SPLINE
SPL {X  -151.875, Y  +721.838, Z    +0.000, E1   -27.241, E3 +55166.889}
SPL {X  -157.803, Y  +697.921, Z    +0.000, E1   -15.861, E3 +55182.756}
SPL {X  -159.710, Y  +681.128, Z    +0.000, E1    -6.465, E3 +55187.890}
SPL {X  -159.999, Y  +671.996, Z    +0.000, E1    -0.411, E3 +55189.220}
SPL {X  -160.000, Y  +665.132, Z    +0.000, E1    +5.902, E3 +55190.030}
SPL {X  -160.000, Y  +655.952, Z    +0.000, E1   +16.601, E3 +55192.025}
SPL {X  -160.000, Y  +643.612, Z    +0.000, E1   +29.091, E3 +55196.997}
SPL {X  -160.000, Y  +606.346, Z    +0.000, E1   +46.235, E3 +55224.805}
SPL {X  -160.000, Y  +564.751, Z    +0.000, E1   +49.682, E3 +55279.976}
SPL {X  -160.000, Y  +555.844, Z    +0.000, E1   +49.673, E3 +55296.057}
SPL {X  -160.000, Y  +545.889, Z    +0.000, E1   +49.702, E3 +55313.956}
SPL {X  -160.000, Y  +535.482, Z    +0.000, E1   +49.684, E3 +55332.755}
SPL {X  -160.000, Y  +526.440, Z    +0.000, E1   +49.666, E3 +55349.088}
SPL {X  -160.000, Y  +518.889, Z    +0.000, E1   +49.624, E3 +55362.913}
ENDSPLINE

SPLINE
SPL {X  -160.000, Y  +548.948, Z    +0.000, E1   +36.551, E3 +55372.601}
ENDSPLINE

SPLINE
SPL {X  -160.000, Y  +541.880, Z    +0.000, E1   +37.562, E3 +55386.380}
SPL {X  -160.000, Y  +532.200, Z    +0.000, E1   +38.842, E3 +55404.721}
SPL {X  -160.000, Y  +523.085, Z    +0.000, E1   +39.970, E3 +55421.412}
SPL {X  -160.000, Y  +513.603, Z    +0.000, E1   +41.139, E3 +55437.996}
SPL {X  -160.000, Y  +503.235, Z    +0.000, E1   +42.462, E3 +55454.704}
SPL {X  -160.000, Y  +493.516, Z    +0.000, E1   +43.493, E3 +55470.749}
SPL {X  -160.000, Y  +483.478, Z    +0.000, E1   +44.599, E3 +55486.207}
SPL {X  -160.000, Y  +473.020, Z    +0.000, E1   +45.665, E3 +55502.037}
SPL {X  -160.000, Y  +461.024, Z    +0.000, E1   +46.836, E3 +55519.512}
SPL {X  -160.000, Y  +448.988, Z    +0.000, E1   +48.043, E3 +55535.774}
SPL {X  -160.000, Y  +439.029, Z    +0.000, E1   +48.623, E3 +55551.181}
SPL {X  -160.000, Y  +429.710, Z    +0.000, E1   +48.622, E3 +55568.628}
SPL {X  -160.000, Y  +420.891, Z    +0.000, E1   +48.613, E3 +55585.153}
SPL {X  -160.000, Y  +412.565, Z    +0.000, E1   +48.611, E3 +55600.718}
SPL {X  -160.000, Y  +404.943, Z    +0.000, E1   +48.601, E3 +55615.021}
SPL {X  -160.000, Y  +395.837, Z    +0.000, E1   +48.634, E3 +55632.010}
SPL {X  -159.987, Y  +386.768, Z    +0.000, E1   +48.609, E3 +55649.015}
SPL {X  -159.620, Y  +377.782, Z    +0.000, E1   +48.569, E3 +55666.183}
SPL {X  -158.761, Y  +368.924, Z    +0.000, E1   +48.401, E3 +55683.710}
SPL {X  -157.560, Y  +360.964, Z    +0.000, E1   +48.177, E3 +55699.881}
SPL {X  -156.187, Y  +354.076, Z    +0.000, E1   +47.920, E3 +55714.214}
SPL {X  -154.507, Y  +347.236, Z    +0.000, E1   +47.623, E3 +55728.742}
SPL {X  -152.108, Y  +339.169, Z    +0.000, E1   +47.215, E3 +55746.219}
SPL {X  -149.264, Y  +331.177, Z    +0.000, E1   +46.657, E3 +55764.018}
SPL {X  -146.675, Y  +324.875, Z    +0.000, E1   +46.130, E3 +55778.371}
SPL {X  -140.793, Y  +312.792, Z    +0.000, E1   +40.077, E3 +55852.614}
ENDSPLINE

SPLINE
SPL {X  -154.674, Y  +347.860, Z    +0.000, E1   +23.016, E3 +55922.757}
SPL {X  -159.179, Y  +372.617, Z    +0.000, E1   +10.186, E3 +55935.406}
SPL {X  -159.924, Y  +383.861, Z    +0.000, E1    +3.320, E3 +55938.028}
SPL {X  -160.000, Y  +389.631, Z    +0.000, E1    -0.873, E3 +55938.744}
SPL {X  -160.000, Y  +394.628, Z    +0.000, E1    -5.657, E3 +55939.420}
SPL {X  -160.000, Y  +401.354, Z    +0.000, E1   -13.067, E3 +55940.811}
SPL {X  -160.000, Y  +413.710, Z    +0.000, E1   -25.976, E3 +55945.603}
SPL {X  -160.000, Y  +449.556, Z    +0.000, E1   -44.518, E3 +55971.645}
SPL {X  -160.000, Y  +494.814, Z    +0.000, E1   -49.280, E3 +56029.994}
SPL {X  -160.000, Y  +504.699, Z    +0.000, E1   -49.282, E3 +56048.074}
SPL {X  -160.000, Y  +515.266, Z    +0.000, E1   -49.291, E3 +56067.388}
SPL {X  -160.000, Y  +526.314, Z    +0.000, E1   -49.296, E3 +56087.617}
SPL {X  -160.000, Y  +536.842, Z    +0.000, E1   -49.263, E3 +56106.943}
SPL {X  -160.000, Y  +547.071, Z    +0.000, E1   -49.286, E3 +56125.620}
SPL {X  -160.000, Y  +558.279, Z    +0.000, E1   -49.288, E3 +56146.124}
SPL {X  -160.000, Y  +568.309, Z    +0.000, E1   -49.259, E3 +56164.519}
SPL {X  -160.000, Y  +579.695, Z    +0.000, E1   -49.320, E3 +56185.249}
SPL {X  -160.000, Y  +592.166, Z    +0.000, E1   -49.294, E3 +56208.109}
SPL {X  -160.000, Y  +603.260, Z    +0.000, E1   -49.285, E3 +56228.434}
SPL {X  -160.000, Y  +615.079, Z    +0.000, E1   -49.301, E3 +56250.046}
SPL {X  -160.000, Y  +627.012, Z    +0.000, E1   -49.289, E3 +56271.898}
SPL {X  -160.000, Y  +638.544, Z    +0.000, E1   -49.285, E3 +56293.009}
SPL {X  -160.000, Y  +649.673, Z    +0.000, E1   -49.278, E3 +56313.382}
SPL {X  -160.000, Y  +661.315, Z    +0.000, E1   -49.297, E3 +56334.652}
SPL {X  -159.993, Y  +672.984, Z    +0.000, E1   -49.282, E3 +56356.043}
SPL {X  -159.528, Y  +683.783, Z    +0.000, E1   -49.201, E3 +56376.297}
SPL {X  -158.288, Y  +694.841, Z    +0.000, E1   -49.005, E3 +56397.811}
SPL {X  -156.479, Y  +704.881, Z    +0.000, E1   -48.644, E3 +56418.125}
SPL {X  -154.000, Y  +714.904, Z    +0.000, E1   -48.243, E3 +56438.934}
SPL {X  -150.967, Y  +724.498, Z    +0.000, E1   -47.642, E3 +56459.599}
SPL {X  -147.384, Y  +733.774, Z    +0.000, E1   -47.000, E3 +56480.072}
SPL {X  -139.301, Y  +750.209, Z    +0.000, E1   -41.935, E3 +56551.253}
ENDSPLINE

SPLINE
SPL {X  -151.875, Y  +721.838, Z    +0.000, E1   -27.241, E3 +56628.423}
SPL {X  -157.803, Y  +697.921, Z    +0.000, E1   -15.861, E3 +56644.290}
SPL {X  -159.710, Y  +681.128, Z    +0.000, E1    -6.465, E3 +56649.424}
SPL {X  -159.999, Y  +671.996, Z    +0.000, E1    -0.411, E3 +56650.754}
SPL {X  -160.000, Y  +665.132, Z    +0.000, E1    +5.902, E3 +56651.564}
SPL {X  -160.000, Y  +655.952, Z    +0.000, E1   +16.601, E3 +56653.560}
SPL {X  -160.000, Y  +643.612, Z    +0.000, E1   +29.091, E3 +56658.531}
SPL {X  -160.000, Y  +606.346, Z    +0.000, E1   +46.235, E3 +56686.339}
SPL {X  -160.000, Y  +564.751, Z    +0.000, E1   +49.682, E3 +56741.511}
SPL {X  -160.000, Y  +555.844, Z    +0.000, E1   +49.673, E3 +56757.591}
SPL {X  -160.000, Y  +545.889, Z    +0.000, E1   +49.702, E3 +56775.490}
SPL {X  -160.000, Y  +535.482, Z    +0.000, E1   +49.684, E3 +56794.289}
SPL {X  -160.000, Y  +526.440, Z    +0.000, E1   +49.666, E3 +56810.623}
SPL {X  -160.000, Y  +518.889, Z    +0.000, E1   +49.624, E3 +56824.447}
ENDSPLINE

SPLINE
SPL {X  -160.000, Y  +548.948, Z    +0.000, E1   +36.551, E3 +56834.136}
ENDSPLINE

SPLINE
SPL {X  -160.000, Y  +541.880, Z    +0.000, E1   +37.562, E3 +56847.914}
SPL {X  -160.000, Y  +532.200, Z    +0.000, E1   +38.842, E3 +56866.255}
SPL {X  -160.000, Y  +523.085, Z    +0.000, E1   +39.970, E3 +56882.946}
SPL {X  -160.000, Y  +513.603, Z    +0.000, E1   +41.139, E3 +56899.530}
SPL {X  -160.000, Y  +503.235, Z    +0.000, E1   +42.462, E3 +56916.238}
SPL {X  -160.000, Y  +493.516, Z    +0.000, E1   +43.493, E3 +56932.283}
SPL {X  -160.000, Y  +483.478, Z    +0.000, E1   +44.599, E3 +56947.741}
SPL {X  -160.000, Y  +473.020, Z    +0.000, E1   +45.665, E3 +56963.571}
SPL {X  -160.000, Y  +461.024, Z    +0.000, E1   +46.836, E3 +56981.046}
SPL {X  -160.000, Y  +448.988, Z    +0.000, E1   +48.043, E3 +56997.308}
SPL {X  -160.000, Y  +439.029, Z    +0.000, E1   +48.623, E3 +57012.715}
SPL {X  -160.000, Y  +429.710, Z    +0.000, E1   +48.622, E3 +57030.162}
SPL {X  -160.000, Y  +420.891, Z    +0.000, E1   +48.613, E3 +57046.687}
SPL {X  -160.000, Y  +412.565, Z    +0.000, E1   +48.611, E3 +57062.253}
SPL {X  -160.000, Y  +404.943, Z    +0.000, E1   +48.601, E3 +57076.555}
SPL {X  -160.000, Y  +395.837, Z    +0.000, E1   +48.634, E3 +57093.545}
SPL {X  -159.987, Y  +386.768, Z    +0.000, E1   +48.609, E3 +57110.549}
SPL {X  -159.620, Y  +377.782, Z    +0.000, E1   +48.569, E3 +57127.717}
SPL {X  -158.761, Y  +368.924, Z    +0.000, E1   +48.401, E3 +57145.244}
SPL {X  -157.560, Y  +360.964, Z    +0.000, E1   +48.177, E3 +57161.415}
SPL {X  -156.187, Y  +354.076, Z    +0.000, E1   +47.920, E3 +57175.748}
SPL {X  -154.507, Y  +347.236, Z    +0.000, E1   +47.623, E3 +57190.276}
SPL {X  -152.108, Y  +339.169, Z    +0.000, E1   +47.215, E3 +57207.753}
SPL {X  -149.264, Y  +331.177, Z    +0.000, E1   +46.657, E3 +57225.552}
SPL {X  -146.675, Y  +324.875, Z    +0.000, E1   +46.130, E3 +57239.905}
SPL {X  -140.793, Y  +312.792, Z    +0.000, E1   +40.077, E3 +57314.148}
ENDSPLINE

SPLINE
SPL {X  -154.674, Y  +347.860, Z    +0.000, E1   +23.016, E3 +57384.291}
SPL {X  -159.179, Y  +372.617, Z    +0.000, E1   +10.186, E3 +57396.940}
SPL {X  -159.924, Y  +383.861, Z    +0.000, E1    +3.320, E3 +57399.562}
SPL {X  -160.000, Y  +389.631, Z    +0.000, E1    -0.873, E3 +57400.278}
SPL {X  -160.000, Y  +394.628, Z    +0.000, E1    -5.657, E3 +57400.954}
SPL {X  -160.000, Y  +401.354, Z    +0.000, E1   -13.067, E3 +57402.345}
SPL {X  -160.000, Y  +413.710, Z    +0.000, E1   -25.976, E3 +57407.137}
SPL {X  -160.000, Y  +449.556, Z    +0.000, E1   -44.518, E3 +57433.179}
SPL {X  -160.000, Y  +494.814, Z    +0.000, E1   -49.280, E3 +57491.529}
SPL {X  -160.000, Y  +504.699, Z    +0.000, E1   -49.282, E3 +57509.608}
SPL {X  -160.000, Y  +515.266, Z    +0.000, E1   -49.291, E3 +57528.922}
SPL {X  -160.000, Y  +526.314, Z    +0.000, E1   -49.296, E3 +57549.151}
SPL {X  -160.000, Y  +536.842, Z    +0.000, E1   -49.263, E3 +57568.477}
SPL {X  -160.000, Y  +547.071, Z    +0.000, E1   -49.286, E3 +57587.154}
SPL {X  -160.000, Y  +558.279, Z    +0.000, E1   -49.288, E3 +57607.658}
SPL {X  -160.000, Y  +568.309, Z    +0.000, E1   -49.259, E3 +57626.053}
SPL {X  -160.000, Y  +579.695, Z    +0.000, E1   -49.320, E3 +57646.784}
SPL {X  -160.000, Y  +592.166, Z    +0.000, E1   -49.294, E3 +57669.643}
SPL {X  -160.000, Y  +603.260, Z    +0.000, E1   -49.285, E3 +57689.968}
SPL {X  -160.000, Y  +615.079, Z    +0.000, E1   -49.301, E3 +57711.580}
SPL {X  -160.000, Y  +627.012, Z    +0.000, E1   -49.289, E3 +57733.432}
SPL {X  -160.000, Y  +638.544, Z    +0.000, E1   -49.285, E3 +57754.543}
SPL {X  -160.000, Y  +649.673, Z    +0.000, E1   -49.278, E3 +57774.916}
SPL {X  -160.000, Y  +661.315, Z    +0.000, E1   -49.297, E3 +57796.186}
SPL {X  -159.993, Y  +672.984, Z    +0.000, E1   -49.282, E3 +57817.577}
SPL {X  -159.528, Y  +683.783, Z    +0.000, E1   -49.201, E3 +57837.832}
SPL {X  -158.288, Y  +694.841, Z    +0.000, E1   -49.005, E3 +57859.345}
SPL {X  -156.479, Y  +704.881, Z    +0.000, E1   -48.644, E3 +57879.659}
SPL {X  -154.000, Y  +714.904, Z    +0.000, E1   -48.243, E3 +57900.468}
SPL {X  -150.967, Y  +724.498, Z    +0.000, E1   -47.642, E3 +57921.133}
SPL {X  -147.384, Y  +733.774, Z    +0.000, E1   -47.000, E3 +57941.606}
SPL {X  -139.301, Y  +750.209, Z    +0.000, E1   -41.935, E3 +58012.787}
ENDSPLINE

SPLINE
SPL {X  -151.875, Y  +721.838, Z    +0.000, E1   -27.241, E3 +58089.958}
SPL {X  -157.803, Y  +697.921, Z    +0.000, E1   -15.861, E3 +58105.825}
SPL {X  -159.710, Y  +681.128, Z    +0.000, E1    -6.465, E3 +58110.958}
SPL {X  -159.999, Y  +671.996, Z    +0.000, E1    -0.411, E3 +58112.288}
SPL {X  -160.000, Y  +665.132, Z    +0.000, E1    +5.902, E3 +58113.098}
SPL {X  -160.000, Y  +655.952, Z    +0.000, E1   +16.601, E3 +58115.094}
SPL {X  -160.000, Y  +643.612, Z    +0.000, E1   +29.091, E3 +58120.065}
SPL {X  -160.000, Y  +606.346, Z    +0.000, E1   +46.235, E3 +58147.873}
SPL {X  -160.000, Y  +564.751, Z    +0.000, E1   +49.682, E3 +58203.045}
SPL {X  -160.000, Y  +555.844, Z    +0.000, E1   +49.673, E3 +58219.125}
SPL {X  -160.000, Y  +545.889, Z    +0.000, E1   +49.702, E3 +58237.024}
SPL {X  -160.000, Y  +535.482, Z    +0.000, E1   +49.684, E3 +58255.824}
SPL {X  -160.000, Y  +526.440, Z    +0.000, E1   +49.666, E3 +58272.157}
SPL {X  -160.000, Y  +518.889, Z    +0.000, E1   +49.624, E3 +58285.981}
ENDSPLINE

SPLINE
SPL {X  -160.000, Y  +548.948, Z    +0.000, E1   +36.551, E3 +58295.670}
ENDSPLINE

SPLINE
SPL {X  -160.000, Y  +541.880, Z    +0.000, E1   +37.562, E3 +58309.448}
SPL {X  -160.000, Y  +532.200, Z    +0.000, E1   +38.842, E3 +58327.790}
SPL {X  -160.000, Y  +523.085, Z    +0.000, E1   +39.970, E3 +58344.480}
SPL {X  -160.000, Y  +513.603, Z    +0.000, E1   +41.139, E3 +58361.064}
SPL {X  -160.000, Y  +503.235, Z    +0.000, E1   +42.462, E3 +58377.772}
SPL {X  -160.000, Y  +493.516, Z    +0.000, E1   +43.493, E3 +58393.817}
SPL {X  -160.000, Y  +483.478, Z    +0.000, E1   +44.599, E3 +58409.275}
SPL {X  -160.000, Y  +473.020, Z    +0.000, E1   +45.665, E3 +58425.105}
SPL {X  -160.000, Y  +461.024, Z    +0.000, E1   +46.836, E3 +58442.580}
SPL {X  -160.000, Y  +448.988, Z    +0.000, E1   +48.043, E3 +58458.842}
SPL {X  -160.000, Y  +439.029, Z    +0.000, E1   +48.623, E3 +58474.250}
SPL {X  -160.000, Y  +429.710, Z    +0.000, E1   +48.622, E3 +58491.696}
SPL {X  -160.000, Y  +420.891, Z    +0.000, E1   +48.613, E3 +58508.221}
SPL {X  -160.000, Y  +412.565, Z    +0.000, E1   +48.611, E3 +58523.787}
SPL {X  -160.000, Y  +404.943, Z    +0.000, E1   +48.601, E3 +58538.089}
SPL {X  -160.000, Y  +395.837, Z    +0.000, E1   +48.634, E3 +58555.079}
SPL {X  -159.987, Y  +386.768, Z    +0.000, E1   +48.609, E3 +58572.083}
SPL {X  -159.620, Y  +377.782, Z    +0.000, E1   +48.569, E3 +58589.251}
SPL {X  -158.761, Y  +368.924, Z    +0.000, E1   +48.401, E3 +58606.778}
SPL {X  -157.560, Y  +360.964, Z    +0.000, E1   +48.177, E3 +58622.950}
SPL {X  -156.187, Y  +354.076, Z    +0.000, E1   +47.920, E3 +58637.282}
SPL {X  -154.507, Y  +347.236, Z    +0.000, E1   +47.623, E3 +58651.810}
SPL {X  -152.108, Y  +339.169, Z    +0.000, E1   +47.215, E3 +58669.288}
SPL {X  -149.264, Y  +331.177, Z    +0.000, E1   +46.657, E3 +58687.086}
SPL {X  -146.675, Y  +324.875, Z    +0.000, E1   +46.130, E3 +58701.439}
SPL {X  -140.793, Y  +312.792, Z    +0.000, E1   +40.077, E3 +58775.683}
ENDSPLINE

SPLINE
SPL {X  -154.674, Y  +347.860, Z    +0.000, E1   +23.016, E3 +58845.826}
SPL {X  -159.179, Y  +372.617, Z    +0.000, E1   +10.186, E3 +58858.474}
SPL {X  -159.924, Y  +383.861, Z    +0.000, E1    +3.320, E3 +58861.097}
SPL {X  -160.000, Y  +389.631, Z    +0.000, E1    -0.873, E3 +58861.812}
SPL {X  -160.000, Y  +394.628, Z    +0.000, E1    -5.657, E3 +58862.488}
SPL {X  -160.000, Y  +401.354, Z    +0.000, E1   -13.067, E3 +58863.879}
SPL {X  -160.000, Y  +413.710, Z    +0.000, E1   -25.976, E3 +58868.672}
SPL {X  -160.000, Y  +449.556, Z    +0.000, E1   -44.518, E3 +58894.713}
SPL {X  -160.000, Y  +494.814, Z    +0.000, E1   -49.280, E3 +58953.063}
SPL {X  -160.000, Y  +504.699, Z    +0.000, E1   -49.282, E3 +58971.143}
SPL {X  -160.000, Y  +515.266, Z    +0.000, E1   -49.291, E3 +58990.456}
SPL {X  -160.000, Y  +526.314, Z    +0.000, E1   -49.296, E3 +59010.685}
SPL {X  -160.000, Y  +536.842, Z    +0.000, E1   -49.263, E3 +59030.011}
SPL {X  -160.000, Y  +547.071, Z    +0.000, E1   -49.286, E3 +59048.688}
SPL {X  -160.000, Y  +558.279, Z    +0.000, E1   -49.288, E3 +59069.192}
SPL {X  -160.000, Y  +568.309, Z    +0.000, E1   -49.259, E3 +59087.587}
SPL {X  -160.000, Y  +579.695, Z    +0.000, E1   -49.320, E3 +59108.318}
SPL {X  -160.000, Y  +592.166, Z    +0.000, E1   -49.294, E3 +59131.177}
SPL {X  -160.000, Y  +603.260, Z    +0.000, E1   -49.285, E3 +59151.502}
SPL {X  -160.000, Y  +615.079, Z    +0.000, E1   -49.301, E3 +59173.114}
SPL {X  -160.000, Y  +627.012, Z    +0.000, E1   -49.289, E3 +59194.967}
SPL {X  -160.000, Y  +638.544, Z    +0.000, E1   -49.285, E3 +59216.077}
SPL {X  -160.000, Y  +649.673, Z    +0.000, E1   -49.278, E3 +59236.450}
SPL {X  -160.000, Y  +661.315, Z    +0.000, E1   -49.297, E3 +59257.720}
SPL {X  -159.993, Y  +672.984, Z    +0.000, E1   -49.282, E3 +59279.111}
SPL {X  -159.528, Y  +683.783, Z    +0.000, E1   -49.201, E3 +59299.366}
SPL {X  -158.288, Y  +694.841, Z    +0.000, E1   -49.005, E3 +59320.879}
SPL {X  -156.479, Y  +704.881, Z    +0.000, E1   -48.644, E3 +59341.193}
SPL {X  -154.000, Y  +714.904, Z    +0.000, E1   -48.243, E3 +59362.002}
SPL {X  -150.967, Y  +724.498, Z    +0.000, E1   -47.642, E3 +59382.668}
SPL {X  -147.384, Y  +733.774, Z    +0.000, E1   -47.000, E3 +59403.140}
SPL {X  -139.301, Y  +750.209, Z    +0.000, E1   -41.935, E3 +59474.321}
ENDSPLINE

SPLINE
SPL {X  -151.875, Y  +721.838, Z    +0.000, E1   -27.241, E3 +59551.492}
SPL {X  -157.803, Y  +697.921, Z    +0.000, E1   -15.861, E3 +59567.359}
SPL {X  -159.710, Y  +681.128, Z    +0.000, E1    -6.465, E3 +59572.492}
SPL {X  -159.999, Y  +671.996, Z    +0.000, E1    -0.411, E3 +59573.823}
SPL {X  -160.000, Y  +665.132, Z    +0.000, E1    +5.902, E3 +59574.633}
SPL {X  -160.000, Y  +655.952, Z    +0.000, E1   +16.601, E3 +59576.628}
SPL {X  -160.000, Y  +643.612, Z    +0.000, E1   +29.091, E3 +59581.599}
SPL {X  -160.000, Y  +606.346, Z    +0.000, E1   +46.235, E3 +59609.407}
SPL {X  -160.000, Y  +564.751, Z    +0.000, E1   +49.682, E3 +59664.579}
SPL {X  -160.000, Y  +555.844, Z    +0.000, E1   +49.673, E3 +59680.659}
SPL {X  -160.000, Y  +545.889, Z    +0.000, E1   +49.702, E3 +59698.558}
SPL {X  -160.000, Y  +535.482, Z    +0.000, E1   +49.684, E3 +59717.358}
SPL {X  -160.000, Y  +526.440, Z    +0.000, E1   +49.666, E3 +59733.691}
SPL {X  -160.000, Y  +518.889, Z    +0.000, E1   +49.624, E3 +59747.515}
ENDSPLINE

SPLINE
SPL {X  -160.000, Y  +548.948, Z    +0.000, E1   +36.551, E3 +59757.204}
ENDSPLINE

SPLINE
SPL {X  -160.000, Y  +541.880, Z    +0.000, E1   +37.562, E3 +59770.982}
SPL {X  -160.000, Y  +532.200, Z    +0.000, E1   +38.842, E3 +59789.324}
SPL {X  -160.000, Y  +523.085, Z    +0.000, E1   +39.970, E3 +59806.014}
SPL {X  -160.000, Y  +513.603, Z    +0.000, E1   +41.139, E3 +59822.598}
SPL {X  -160.000, Y  +503.235, Z    +0.000, E1   +42.462, E3 +59839.306}
SPL {X  -160.000, Y  +493.516, Z    +0.000, E1   +43.493, E3 +59855.351}
SPL {X  -160.000, Y  +483.478, Z    +0.000, E1   +44.599, E3 +59870.809}
SPL {X  -160.000, Y  +473.020, Z    +0.000, E1   +45.665, E3 +59886.639}
SPL {X  -160.000, Y  +461.024, Z    +0.000, E1   +46.836, E3 +59904.114}
SPL {X  -160.000, Y  +448.988, Z    +0.000, E1   +48.043, E3 +59920.376}
SPL {X  -160.000, Y  +439.029, Z    +0.000, E1   +48.623, E3 +59935.784}
SPL {X  -160.000, Y  +429.710, Z    +0.000, E1   +48.622, E3 +59953.230}
SPL {X  -160.000, Y  +420.891, Z    +0.000, E1   +48.613, E3 +59969.755}
SPL {X  -160.000, Y  +412.565, Z    +0.000, E1   +48.611, E3 +59985.321}
SPL {X  -160.000, Y  +404.943, Z    +0.000, E1   +48.601, E3 +59999.623}
SPL {X  -160.000, Y  +395.837, Z    +0.000, E1   +48.634, E3 +60016.613}
SPL {X  -159.987, Y  +386.768, Z    +0.000, E1   +48.609, E3 +60033.617}
SPL {X  -159.620, Y  +377.782, Z    +0.000, E1   +48.569, E3 +60050.785}
SPL {X  -158.761, Y  +368.924, Z    +0.000, E1   +48.401, E3 +60068.312}
SPL {X  -157.560, Y  +360.964, Z    +0.000, E1   +48.177, E3 +60084.484}
SPL {X  -156.187, Y  +354.076, Z    +0.000, E1   +47.920, E3 +60098.816}
SPL {X  -154.507, Y  +347.236, Z    +0.000, E1   +47.623, E3 +60113.344}
SPL {X  -152.108, Y  +339.169, Z    +0.000, E1   +47.215, E3 +60130.822}
SPL {X  -149.264, Y  +331.177, Z    +0.000, E1   +46.657, E3 +60148.621}
SPL {X  -146.675, Y  +324.875, Z    +0.000, E1   +46.130, E3 +60162.973}
SPL {X  -140.793, Y  +312.792, Z    +0.000, E1   +40.077, E3 +60237.217}
ENDSPLINE

SPLINE
SPL {X  -154.674, Y  +347.860, Z    +0.000, E1   +23.016, E3 +60307.360}
SPL {X  -159.179, Y  +372.617, Z    +0.000, E1   +10.186, E3 +60320.008}
SPL {X  -159.924, Y  +383.861, Z    +0.000, E1    +3.320, E3 +60322.631}
SPL {X  -160.000, Y  +389.631, Z    +0.000, E1    -0.873, E3 +60323.346}
SPL {X  -160.000, Y  +394.628, Z    +0.000, E1    -5.657, E3 +60324.022}
SPL {X  -160.000, Y  +401.354, Z    +0.000, E1   -13.067, E3 +60325.413}
SPL {X  -160.000, Y  +413.710, Z    +0.000, E1   -25.976, E3 +60330.206}
SPL {X  -160.000, Y  +449.556, Z    +0.000, E1   -44.518, E3 +60356.247}
SPL {X  -160.000, Y  +494.814, Z    +0.000, E1   -49.280, E3 +60414.597}
SPL {X  -160.000, Y  +504.699, Z    +0.000, E1   -49.282, E3 +60432.677}
SPL {X  -160.000, Y  +515.266, Z    +0.000, E1   -49.291, E3 +60451.990}
SPL {X  -160.000, Y  +526.314, Z    +0.000, E1   -49.296, E3 +60472.220}
SPL {X  -160.000, Y  +536.842, Z    +0.000, E1   -49.263, E3 +60491.546}
SPL {X  -160.000, Y  +547.071, Z    +0.000, E1   -49.286, E3 +60510.222}
SPL {X  -160.000, Y  +558.279, Z    +0.000, E1   -49.288, E3 +60530.726}
SPL {X  -160.000, Y  +568.309, Z    +0.000, E1   -49.259, E3 +60549.121}
SPL {X  -160.000, Y  +579.695, Z    +0.000, E1   -49.320, E3 +60569.852}
SPL {X  -160.000, Y  +592.166, Z    +0.000, E1   -49.294, E3 +60592.712}
SPL {X  -160.000, Y  +603.260, Z    +0.000, E1   -49.285, E3 +60613.036}
SPL {X  -160.000, Y  +615.079, Z    +0.000, E1   -49.301, E3 +60634.648}
SPL {X  -160.000, Y  +627.012, Z    +0.000, E1   -49.289, E3 +60656.501}
SPL {X  -160.000, Y  +638.544, Z    +0.000, E1   -49.285, E3 +60677.611}
SPL {X  -160.000, Y  +649.673, Z    +0.000, E1   -49.278, E3 +60697.984}
SPL {X  -160.000, Y  +661.315, Z    +0.000, E1   -49.297, E3 +60719.255}
SPL {X  -159.993, Y  +672.984, Z    +0.000, E1   -49.282, E3 +60740.645}
SPL {X  -159.528, Y  +683.783, Z    +0.000, E1   -49.201, E3 +60760.900}
SPL {X  -158.288, Y  +694.841, Z    +0.000, E1   -49.005, E3 +60782.413}
SPL {X  -156.479, Y  +704.881, Z    +0.000, E1   -48.644, E3 +60802.727}
SPL {X  -154.000, Y  +714.904, Z    +0.000, E1   -48.243, E3 +60823.536}
SPL {X  -150.967, Y  +724.498, Z    +0.000, E1   -47.642, E3 +60844.202}
SPL {X  -147.384, Y  +733.774, Z    +0.000, E1   -47.000, E3 +60864.675}
SPL {X  -139.301, Y  +750.209, Z    +0.000, E1   -41.935, E3 +60935.856}
ENDSPLINE

SPLINE
SPL {X  -151.875, Y  +721.838, Z    +0.000, E1   -27.241, E3 +61013.026}
SPL {X  -157.803, Y  +697.921, Z    +0.000, E1   -15.861, E3 +61028.893}
SPL {X  -159.710, Y  +681.128, Z    +0.000, E1    -6.465, E3 +61034.026}
SPL {X  -159.999, Y  +671.996, Z    +0.000, E1    -0.411, E3 +61035.357}
SPL {X  -160.000, Y  +665.132, Z    +0.000, E1    +5.902, E3 +61036.167}
SPL {X  -160.000, Y  +655.952, Z    +0.000, E1   +16.601, E3 +61038.162}
SPL {X  -160.000, Y  +643.612, Z    +0.000, E1   +29.091, E3 +61043.133}
SPL {X  -160.000, Y  +606.346, Z    +0.000, E1   +46.235, E3 +61070.941}
SPL {X  -160.000, Y  +564.751, Z    +0.000, E1   +49.682, E3 +61126.113}
SPL {X  -160.000, Y  +555.844, Z    +0.000, E1   +49.673, E3 +61142.194}
SPL {X  -160.000, Y  +545.889, Z    +0.000, E1   +49.702, E3 +61160.092}
SPL {X  -160.000, Y  +535.482, Z    +0.000, E1   +49.684, E3 +61178.892}
SPL {X  -160.000, Y  +526.440, Z    +0.000, E1   +49.666, E3 +61195.225}
SPL {X  -160.000, Y  +518.889, Z    +0.000, E1   +49.624, E3 +61209.049}
ENDSPLINE

SPLINE
SPL {X  -160.000, Y  +548.948, Z    +0.000, E1   +36.551, E3 +61218.738}
ENDSPLINE

SPLINE
SPL {X  -160.000, Y  +541.880, Z    +0.000, E1   +37.562, E3 +61232.516}
SPL {X  -160.000, Y  +532.200, Z    +0.000, E1   +38.842, E3 +61250.858}
SPL {X  -160.000, Y  +523.085, Z    +0.000, E1   +39.970, E3 +61267.548}
SPL {X  -160.000, Y  +513.603, Z    +0.000, E1   +41.139, E3 +61284.132}
SPL {X  -160.000, Y  +503.235, Z    +0.000, E1   +42.462, E3 +61300.840}
SPL {X  -160.000, Y  +493.516, Z    +0.000, E1   +43.493, E3 +61316.885}
SPL {X  -160.000, Y  +483.478, Z    +0.000, E1   +44.599, E3 +61332.343}
SPL {X  -160.000, Y  +473.020, Z    +0.000, E1   +45.665, E3 +61348.173}
SPL {X  -160.000, Y  +461.024, Z    +0.000, E1   +46.836, E3 +61365.648}
SPL {X  -160.000, Y  +448.988, Z    +0.000, E1   +48.043, E3 +61381.910}
SPL {X  -160.000, Y  +439.029, Z    +0.000, E1   +48.623, E3 +61397.318}
SPL {X  -160.000, Y  +429.710, Z    +0.000, E1   +48.622, E3 +61414.765}
SPL {X  -160.000, Y  +420.891, Z    +0.000, E1   +48.613, E3 +61431.289}
SPL {X  -160.000, Y  +412.565, Z    +0.000, E1   +48.611, E3 +61446.855}
SPL {X  -160.000, Y  +404.943, Z    +0.000, E1   +48.601, E3 +61461.157}
SPL {X  -160.000, Y  +395.837, Z    +0.000, E1   +48.634, E3 +61478.147}
SPL {X  -159.987, Y  +386.768, Z    +0.000, E1   +48.609, E3 +61495.151}
SPL {X  -159.620, Y  +377.782, Z    +0.000, E1   +48.569, E3 +61512.319}
SPL {X  -158.761, Y  +368.924, Z    +0.000, E1   +48.401, E3 +61529.846}
SPL {X  -157.560, Y  +360.964, Z    +0.000, E1   +48.177, E3 +61546.018}
SPL {X  -156.187, Y  +354.076, Z    +0.000, E1   +47.920, E3 +61560.351}
SPL {X  -154.507, Y  +347.236, Z    +0.000, E1   +47.623, E3 +61574.878}
SPL {X  -152.108, Y  +339.169, Z    +0.000, E1   +47.215, E3 +61592.356}
SPL {X  -149.264, Y  +331.177, Z    +0.000, E1   +46.657, E3 +61610.155}
SPL {X  -146.675, Y  +324.875, Z    +0.000, E1   +46.130, E3 +61624.508}
SPL {X  -140.793, Y  +312.792, Z    +0.000, E1   +40.077, E3 +61698.751}
ENDSPLINE

SPLINE
SPL {X  -154.674, Y  +347.860, Z    +0.000, E1   +23.016, E3 +61768.894}
SPL {X  -159.179, Y  +372.617, Z    +0.000, E1   +10.186, E3 +61781.542}
SPL {X  -159.924, Y  +383.861, Z    +0.000, E1    +3.320, E3 +61784.165}
SPL {X  -160.000, Y  +389.631, Z    +0.000, E1    -0.873, E3 +61784.881}
SPL {X  -160.000, Y  +394.628, Z    +0.000, E1    -5.657, E3 +61785.556}
SPL {X  -160.000, Y  +401.354, Z    +0.000, E1   -13.067, E3 +61786.947}
SPL {X  -160.000, Y  +413.710, Z    +0.000, E1   -25.976, E3 +61791.740}
SPL {X  -160.000, Y  +449.556, Z    +0.000, E1   -44.518, E3 +61817.781}
SPL {X  -160.000, Y  +494.814, Z    +0.000, E1   -49.280, E3 +61876.131}
SPL {X  -160.000, Y  +504.699, Z    +0.000, E1   -49.282, E3 +61894.211}
SPL {X  -160.000, Y  +515.266, Z    +0.000, E1   -49.291, E3 +61913.525}
SPL {X  -160.000, Y  +526.314, Z    +0.000, E1   -49.296, E3 +61933.754}
SPL {X  -160.000, Y  +536.842, Z    +0.000, E1   -49.263, E3 +61953.080}
SPL {X  -160.000, Y  +547.071, Z    +0.000, E1   -49.286, E3 +61971.756}
SPL {X  -160.000, Y  +558.279, Z    +0.000, E1   -49.288, E3 +61992.260}
SPL {X  -160.000, Y  +568.309, Z    +0.000, E1   -49.259, E3 +62010.655}
SPL {X  -160.000, Y  +579.695, Z    +0.000, E1   -49.320, E3 +62031.386}
SPL {X  -160.000, Y  +592.166, Z    +0.000, E1   -49.294, E3 +62054.246}
SPL {X  -160.000, Y  +603.260, Z    +0.000, E1   -49.285, E3 +62074.570}
SPL {X  -160.000, Y  +615.079, Z    +0.000, E1   -49.301, E3 +62096.182}
SPL {X  -160.000, Y  +627.012, Z    +0.000, E1   -49.289, E3 +62118.035}
SPL {X  -160.000, Y  +638.544, Z    +0.000, E1   -49.285, E3 +62139.145}
SPL {X  -160.000, Y  +649.673, Z    +0.000, E1   -49.278, E3 +62159.519}
SPL {X  -160.000, Y  +661.315, Z    +0.000, E1   -49.297, E3 +62180.789}
SPL {X  -159.993, Y  +672.984, Z    +0.000, E1   -49.282, E3 +62202.179}
SPL {X  -159.528, Y  +683.783, Z    +0.000, E1   -49.201, E3 +62222.434}
SPL {X  -158.288, Y  +694.841, Z    +0.000, E1   -49.005, E3 +62243.947}
SPL {X  -156.479, Y  +704.881, Z    +0.000, E1   -48.644, E3 +62264.261}
SPL {X  -154.000, Y  +714.904, Z    +0.000, E1   -48.243, E3 +62285.070}
SPL {X  -150.967, Y  +724.498, Z    +0.000, E1   -47.642, E3 +62305.736}
SPL {X  -147.384, Y  +733.774, Z    +0.000, E1   -47.000, E3 +62326.209}
SPL {X  -139.301, Y  +750.209, Z    +0.000, E1   -41.935, E3 +62397.390}
ENDSPLINE

SPLINE
SPL {X  -151.875, Y  +721.838, Z    +0.000, E1   -27.241, E3 +62474.560}
SPL {X  -157.803, Y  +697.921, Z    +0.000, E1   -15.861, E3 +62490.427}
SPL {X  -159.710, Y  +681.128, Z    +0.000, E1    -6.465, E3 +62495.560}
SPL {X  -159.999, Y  +671.996, Z    +0.000, E1    -0.411, E3 +62496.891}
SPL {X  -160.000, Y  +665.132, Z    +0.000, E1    +5.902, E3 +62497.701}
SPL {X  -160.000, Y  +655.952, Z    +0.000, E1   +16.601, E3 +62499.696}
SPL {X  -160.000, Y  +643.612, Z    +0.000, E1   +29.091, E3 +62504.667}
SPL {X  -160.000, Y  +606.346, Z    +0.000, E1   +46.235, E3 +62532.475}
SPL {X  -160.000, Y  +564.751, Z    +0.000, E1   +49.682, E3 +62587.647}
SPL {X  -160.000, Y  +555.844, Z    +0.000, E1   +49.673, E3 +62603.728}
SPL {X  -160.000, Y  +545.889, Z    +0.000, E1   +49.702, E3 +62621.626}
SPL {X  -160.000, Y  +535.482, Z    +0.000, E1   +49.684, E3 +62640.426}
SPL {X  -160.000, Y  +526.440, Z    +0.000, E1   +49.666, E3 +62656.759}
SPL {X  -160.000, Y  +518.889, Z    +0.000, E1   +49.624, E3 +62670.583}
ENDSPLINE

SPLINE
SPL {X  -160.000, Y  +548.948, Z    +0.000, E1   +36.551, E3 +62680.272}
ENDSPLINE

SPLINE
SPL {X  -160.000, Y  +541.880, Z    +0.000, E1   +37.562, E3 +62694.050}
SPL {X  -160.000, Y  +532.200, Z    +0.000, E1   +38.842, E3 +62712.392}
SPL {X  -160.000, Y  +523.085, Z    +0.000, E1   +39.970, E3 +62729.082}
SPL {X  -160.000, Y  +513.603, Z    +0.000, E1   +41.139, E3 +62745.666}
SPL {X  -160.000, Y  +503.235, Z    +0.000, E1   +42.462, E3 +62762.375}
SPL {X  -160.000, Y  +493.516, Z    +0.000, E1   +43.493, E3 +62778.420}
SPL {X  -160.000, Y  +483.478, Z    +0.000, E1   +44.599, E3 +62793.878}
SPL {X  -160.000, Y  +473.020, Z    +0.000, E1   +45.665, E3 +62809.707}
SPL {X  -160.000, Y  +461.024, Z    +0.000, E1   +46.836, E3 +62827.183}
SPL {X  -160.000, Y  +448.988, Z    +0.000, E1   +48.043, E3 +62843.444}
SPL {X  -160.000, Y  +439.029, Z    +0.000, E1   +48.623, E3 +62858.852}
SPL {X  -160.000, Y  +429.710, Z    +0.000, E1   +48.622, E3 +62876.299}
SPL {X  -160.000, Y  +420.891, Z    +0.000, E1   +48.613, E3 +62892.824}
SPL {X  -160.000, Y  +412.565, Z    +0.000, E1   +48.611, E3 +62908.389}
SPL {X  -160.000, Y  +404.943, Z    +0.000, E1   +48.601, E3 +62922.692}
SPL {X  -160.000, Y  +395.837, Z    +0.000, E1   +48.634, E3 +62939.681}
SPL {X  -159.987, Y  +386.768, Z    +0.000, E1   +48.609, E3 +62956.685}
SPL {X  -159.620, Y  +377.782, Z    +0.000, E1   +48.569, E3 +62973.853}
SPL {X  -158.761, Y  +368.924, Z    +0.000, E1   +48.401, E3 +62991.380}
SPL {X  -157.560, Y  +360.964, Z    +0.000, E1   +48.177, E3 +63007.552}
SPL {X  -156.187, Y  +354.076, Z    +0.000, E1   +47.920, E3 +63021.885}
SPL {X  -154.507, Y  +347.236, Z    +0.000, E1   +47.623, E3 +63036.413}
SPL {X  -152.108, Y  +339.169, Z    +0.000, E1   +47.215, E3 +63053.890}
SPL {X  -149.264, Y  +331.177, Z    +0.000, E1   +46.657, E3 +63071.689}
SPL {X  -146.675, Y  +324.875, Z    +0.000, E1   +46.130, E3 +63086.042}
SPL {X  -140.793, Y  +312.792, Z    +0.000, E1   +40.077, E3 +63160.285}
ENDSPLINE

SPLINE
SPL {X  -154.674, Y  +347.860, Z    +0.000, E1   +23.016, E3 +63230.428}
SPL {X  -159.179, Y  +372.617, Z    +0.000, E1   +10.186, E3 +63243.076}
SPL {X  -159.924, Y  +383.861, Z    +0.000, E1    +3.320, E3 +63245.699}
SPL {X  -160.000, Y  +389.631, Z    +0.000, E1    -0.873, E3 +63246.415}
SPL {X  -160.000, Y  +394.628, Z    +0.000, E1    -5.657, E3 +63247.090}
SPL {X  -160.000, Y  +401.354, Z    +0.000, E1   -13.067, E3 +63248.481}
SPL {X  -160.000, Y  +413.710, Z    +0.000, E1   -25.976, E3 +63253.274}
SPL {X  -160.000, Y  +449.556, Z    +0.000, E1   -44.518, E3 +63279.315}
SPL {X  -160.000, Y  +494.814, Z    +0.000, E1   -49.280, E3 +63337.665}
SPL {X  -160.000, Y  +504.699, Z    +0.000, E1   -49.282, E3 +63355.745}
SPL {X  -160.000, Y  +515.266, Z    +0.000, E1   -49.291, E3 +63375.059}
SPL {X  -160.000, Y  +526.314, Z    +0.000, E1   -49.296, E3 +63395.288}
SPL {X  -160.000, Y  +536.842, Z    +0.000, E1   -49.263, E3 +63414.614}
SPL {X  -160.000, Y  +547.071, Z    +0.000, E1   -49.286, E3 +63433.290}
SPL {X  -160.000, Y  +558.279, Z    +0.000, E1   -49.288, E3 +63453.794}
SPL {X  -160.000, Y  +568.309, Z    +0.000, E1   -49.259, E3 +63472.190}
SPL {X  -160.000, Y  +579.695, Z    +0.000, E1   -49.320, E3 +63492.920}
SPL {X  -160.000, Y  +592.166, Z    +0.000, E1   -49.294, E3 +63515.780}
SPL {X  -160.000, Y  +603.260, Z    +0.000, E1   -49.285, E3 +63536.104}
SPL {X  -160.000, Y  +615.079, Z    +0.000, E1   -49.301, E3 +63557.716}
SPL {X  -160.000, Y  +627.012, Z    +0.000, E1   -49.289, E3 +63579.569}
SPL {X  -160.000, Y  +638.544, Z    +0.000, E1   -49.285, E3 +63600.679}
SPL {X  -160.000, Y  +649.673, Z    +0.000, E1   -49.278, E3 +63621.053}
SPL {X  -160.000, Y  +661.315, Z    +0.000, E1   -49.297, E3 +63642.323}
SPL {X  -159.993, Y  +672.984, Z    +0.000, E1   -49.282, E3 +63663.713}
SPL {X  -159.528, Y  +683.783, Z    +0.000, E1   -49.201, E3 +63683.968}
SPL {X  -158.288, Y  +694.841, Z    +0.000, E1   -49.005, E3 +63705.482}
SPL {X  -156.479, Y  +704.881, Z    +0.000, E1   -48.644, E3 +63725.795}
SPL {X  -154.000, Y  +714.904, Z    +0.000, E1   -48.243, E3 +63746.605}
SPL {X  -150.967, Y  +724.498, Z    +0.000, E1   -47.642, E3 +63767.270}
SPL {X  -147.384, Y  +733.774, Z    +0.000, E1   -47.000, E3 +63787.743}
SPL {X  -139.301, Y  +750.209, Z    +0.000, E1   -41.935, E3 +63858.924}
ENDSPLINE

SPLINE
SPL {X  -151.875, Y  +721.838, Z    +0.000, E1   -27.241, E3 +63936.094}
SPL {X  -157.803, Y  +697.921, Z    +0.000, E1   -15.861, E3 +63951.961}
SPL {X  -159.710, Y  +681.128, Z    +0.000, E1    -6.465, E3 +63957.095}
SPL {X  -159.999, Y  +671.996, Z    +0.000, E1    -0.411, E3 +63958.425}
SPL {X  -160.000, Y  +665.132, Z    +0.000, E1    +5.902, E3 +63959.235}
SPL {X  -160.000, Y  +655.952, Z    +0.000, E1   +16.601, E3 +63961.230}
SPL {X  -160.000, Y  +643.612, Z    +0.000, E1   +29.091, E3 +63966.202}
SPL {X  -160.000, Y  +606.346, Z    +0.000, E1   +46.235, E3 +63994.010}
SPL {X  -160.000, Y  +564.751, Z    +0.000, E1   +49.682, E3 +64049.181}
SPL {X  -160.000, Y  +555.844, Z    +0.000, E1   +49.673, E3 +64065.262}
SPL {X  -160.000, Y  +545.889, Z    +0.000, E1   +49.702, E3 +64083.160}
SPL {X  -160.000, Y  +535.482, Z    +0.000, E1   +49.684, E3 +64101.960}
SPL {X  -160.000, Y  +526.440, Z    +0.000, E1   +49.666, E3 +64118.293}
SPL {X  -160.000, Y  +518.889, Z    +0.000, E1   +49.624, E3 +64132.118}
ENDSPLINE

SPLINE
SPL {X  -160.000, Y  +548.948, Z    +0.000, E1   +36.551, E3 +64141.806}
ENDSPLINE

SPLINE
SPL {X  -160.000, Y  +541.880, Z    +0.000, E1   +37.562, E3 +64155.584}
SPL {X  -160.000, Y  +532.200, Z    +0.000, E1   +38.842, E3 +64173.926}
SPL {X  -160.000, Y  +523.085, Z    +0.000, E1   +39.970, E3 +64190.617}
SPL {X  -160.000, Y  +513.603, Z    +0.000, E1   +41.139, E3 +64207.201}
SPL {X  -160.000, Y  +503.235, Z    +0.000, E1   +42.462, E3 +64223.909}
SPL {X  -160.000, Y  +493.516, Z    +0.000, E1   +43.493, E3 +64239.954}
SPL {X  -160.000, Y  +483.478, Z    +0.000, E1   +44.599, E3 +64255.412}
SPL {X  -160.000, Y  +473.020, Z    +0.000, E1   +45.665, E3 +64271.241}
SPL {X  -160.000, Y  +461.024, Z    +0.000, E1   +46.836, E3 +64288.717}
SPL {X  -160.000, Y  +448.988, Z    +0.000, E1   +48.043, E3 +64304.978}
SPL {X  -160.000, Y  +439.029, Z    +0.000, E1   +48.623, E3 +64320.386}
SPL {X  -160.000, Y  +429.710, Z    +0.000, E1   +48.622, E3 +64337.833}
SPL {X  -160.000, Y  +420.891, Z    +0.000, E1   +48.613, E3 +64354.358}
SPL {X  -160.000, Y  +412.565, Z    +0.000, E1   +48.611, E3 +64369.923}
SPL {X  -160.000, Y  +404.943, Z    +0.000, E1   +48.601, E3 +64384.226}
SPL {X  -160.000, Y  +395.837, Z    +0.000, E1   +48.634, E3 +64401.215}
SPL {X  -159.987, Y  +386.768, Z    +0.000, E1   +48.609, E3 +64418.220}
SPL {X  -159.620, Y  +377.782, Z    +0.000, E1   +48.569, E3 +64435.387}
SPL {X  -158.761, Y  +368.924, Z    +0.000, E1   +48.401, E3 +64452.915}
SPL {X  -157.560, Y  +360.964, Z    +0.000, E1   +48.177, E3 +64469.086}
SPL {X  -156.187, Y  +354.076, Z    +0.000, E1   +47.920, E3 +64483.419}
SPL {X  -154.507, Y  +347.236, Z    +0.000, E1   +47.623, E3 +64497.947}
SPL {X  -152.108, Y  +339.169, Z    +0.000, E1   +47.215, E3 +64515.424}
SPL {X  -149.264, Y  +331.177, Z    +0.000, E1   +46.657, E3 +64533.223}
SPL {X  -146.675, Y  +324.875, Z    +0.000, E1   +46.130, E3 +64547.576}
SPL {X  -140.793, Y  +312.792, Z    +0.000, E1   +40.077, E3 +64621.819}
ENDSPLINE

SPLINE
SPL {X  -154.674, Y  +347.860, Z    +0.000, E1   +23.016, E3 +64691.962}
SPL {X  -159.179, Y  +372.617, Z    +0.000, E1   +10.186, E3 +64704.611}
SPL {X  -159.924, Y  +383.861, Z    +0.000, E1    +3.320, E3 +64707.233}
SPL {X  -160.000, Y  +389.631, Z    +0.000, E1    -0.873, E3 +64707.949}
SPL {X  -160.000, Y  +394.628, Z    +0.000, E1    -5.657, E3 +64708.624}
SPL {X  -160.000, Y  +401.354, Z    +0.000, E1   -13.067, E3 +64710.016}
SPL {X  -160.000, Y  +413.710, Z    +0.000, E1   -25.976, E3 +64714.808}
SPL {X  -160.000, Y  +449.556, Z    +0.000, E1   -44.518, E3 +64740.850}
SPL {X  -160.000, Y  +494.814, Z    +0.000, E1   -49.280, E3 +64799.199}
SPL {X  -160.000, Y  +504.699, Z    +0.000, E1   -49.282, E3 +64817.279}
SPL {X  -160.000, Y  +515.266, Z    +0.000, E1   -49.291, E3 +64836.593}
SPL {X  -160.000, Y  +526.314, Z    +0.000, E1   -49.296, E3 +64856.822}
SPL {X  -160.000, Y  +536.842, Z    +0.000, E1   -49.263, E3 +64876.148}
SPL {X  -160.000, Y  +547.071, Z    +0.000, E1   -49.286, E3 +64894.825}
SPL {X  -160.000, Y  +558.279, Z    +0.000, E1   -49.288, E3 +64915.329}
SPL {X  -160.000, Y  +568.309, Z    +0.000, E1   -49.259, E3 +64933.724}
SPL {X  -160.000, Y  +579.695, Z    +0.000, E1   -49.320, E3 +64954.454}
SPL {X  -160.000, Y  +592.166, Z    +0.000, E1   -49.294, E3 +64977.314}
SPL {X  -160.000, Y  +603.260, Z    +0.000, E1   -49.285, E3 +64997.638}
SPL {X  -160.000, Y  +615.079, Z    +0.000, E1   -49.301, E3 +65019.251}
SPL {X  -160.000, Y  +627.012, Z    +0.000, E1   -49.289, E3 +65041.103}
SPL {X  -160.000, Y  +638.544, Z    +0.000, E1   -49.285, E3 +65062.213}
SPL {X  -160.000, Y  +649.673, Z    +0.000, E1   -49.278, E3 +65082.587}
SPL {X  -160.000, Y  +661.315, Z    +0.000, E1   -49.297, E3 +65103.857}
SPL {X  -159.993, Y  +672.984, Z    +0.000, E1   -49.282, E3 +65125.248}
SPL {X  -159.528, Y  +683.783, Z    +0.000, E1   -49.201, E3 +65145.502}
SPL {X  -158.288, Y  +694.841, Z    +0.000, E1   -49.005, E3 +65167.016}
SPL {X  -156.479, Y  +704.881, Z    +0.000, E1   -48.644, E3 +65187.329}
SPL {X  -154.000, Y  +714.904, Z    +0.000, E1   -48.243, E3 +65208.139}
SPL {X  -150.967, Y  +724.498, Z    +0.000, E1   -47.642, E3 +65228.804}
SPL {X  -147.384, Y  +733.774, Z    +0.000, E1   -47.000, E3 +65249.277}
SPL {X  -139.301, Y  +750.209, Z    +0.000, E1   -41.935, E3 +65320.458}
ENDSPLINE

SPLINE
SPL {X  -151.875, Y  +721.838, Z    +0.000, E1   -27.241, E3 +65397.628}
SPL {X  -157.803, Y  +697.921, Z    +0.000, E1   -15.861, E3 +65413.495}
SPL {X  -159.710, Y  +681.128, Z    +0.000, E1    -6.465, E3 +65418.629}
SPL {X  -159.999, Y  +671.996, Z    +0.000, E1    -0.411, E3 +65419.959}
SPL {X  -160.000, Y  +665.132, Z    +0.000, E1    +5.902, E3 +65420.769}
SPL {X  -160.000, Y  +655.952, Z    +0.000, E1   +16.601, E3 +65422.764}
SPL {X  -160.000, Y  +643.612, Z    +0.000, E1   +29.091, E3 +65427.736}
SPL {X  -160.000, Y  +606.346, Z    +0.000, E1   +46.235, E3 +65455.544}
SPL {X  -160.000, Y  +564.751, Z    +0.000, E1   +49.682, E3 +65510.715}
SPL {X  -160.000, Y  +555.844, Z    +0.000, E1   +49.673, E3 +65526.796}
SPL {X  -160.000, Y  +545.889, Z    +0.000, E1   +49.702, E3 +65544.695}
SPL {X  -160.000, Y  +535.482, Z    +0.000, E1   +49.684, E3 +65563.494}
SPL {X  -160.000, Y  +526.440, Z    +0.000, E1   +49.666, E3 +65579.827}
SPL {X  -160.000, Y  +518.889, Z    +0.000, E1   +49.624, E3 +65593.652}
ENDSPLINE

SPLINE
SPL {X  -160.000, Y  +548.948, Z    +0.000, E1   +36.551, E3 +65603.340}
ENDSPLINE

SPLINE
SPL {X  -160.000, Y  +541.880, Z    +0.000, E1   +37.562, E3 +65617.118}
SPL {X  -160.000, Y  +532.200, Z    +0.000, E1   +38.842, E3 +65635.460}
SPL {X  -160.000, Y  +523.085, Z    +0.000, E1   +39.970, E3 +65652.151}
SPL {X  -160.000, Y  +513.603, Z    +0.000, E1   +41.139, E3 +65668.735}
SPL {X  -160.000, Y  +503.235, Z    +0.000, E1   +42.462, E3 +65685.443}
SPL {X  -160.000, Y  +493.516, Z    +0.000, E1   +43.493, E3 +65701.488}
SPL {X  -160.000, Y  +483.478, Z    +0.000, E1   +44.599, E3 +65716.946}
SPL {X  -160.000, Y  +473.020, Z    +0.000, E1   +45.665, E3 +65732.776}
SPL {X  -160.000, Y  +461.024, Z    +0.000, E1   +46.836, E3 +65750.251}
SPL {X  -160.000, Y  +448.988, Z    +0.000, E1   +48.043, E3 +65766.512}
SPL {X  -160.000, Y  +439.029, Z    +0.000, E1   +48.623, E3 +65781.920}
SPL {X  -160.000, Y  +429.710, Z    +0.000, E1   +48.622, E3 +65799.367}
SPL {X  -160.000, Y  +420.891, Z    +0.000, E1   +48.613, E3 +65815.892}
SPL {X  -160.000, Y  +412.565, Z    +0.000, E1   +48.611, E3 +65831.457}
SPL {X  -160.000, Y  +404.943, Z    +0.000, E1   +48.601, E3 +65845.760}
SPL {X  -160.000, Y  +395.837, Z    +0.000, E1   +48.634, E3 +65862.749}
SPL {X  -159.987, Y  +386.768, Z    +0.000, E1   +48.609, E3 +65879.754}
SPL {X  -159.620, Y  +377.782, Z    +0.000, E1   +48.569, E3 +65896.921}
SPL {X  -158.761, Y  +368.924, Z    +0.000, E1   +48.401, E3 +65914.449}
SPL {X  -157.560, Y  +360.964, Z    +0.000, E1   +48.177, E3 +65930.620}
SPL {X  -156.187, Y  +354.076, Z    +0.000, E1   +47.920, E3 +65944.953}
SPL {X  -154.507, Y  +347.236, Z    +0.000, E1   +47.623, E3 +65959.481}
SPL {X  -152.108, Y  +339.169, Z    +0.000, E1   +47.215, E3 +65976.958}
SPL {X  -149.264, Y  +331.177, Z    +0.000, E1   +46.657, E3 +65994.757}
SPL {X  -146.675, Y  +324.875, Z    +0.000, E1   +46.130, E3 +66009.110}
SPL {X  -140.793, Y  +312.792, Z    +0.000, E1   +40.077, E3 +66083.353}
ENDSPLINE

SPLINE
SPL {X  -154.674, Y  +347.860, Z    +0.000, E1   +23.016, E3 +66153.496}
SPL {X  -159.179, Y  +372.617, Z    +0.000, E1   +10.186, E3 +66166.145}
SPL {X  -159.924, Y  +383.861, Z    +0.000, E1    +3.320, E3 +66168.767}
SPL {X  -160.000, Y  +389.631, Z    +0.000, E1    -0.873, E3 +66169.483}
SPL {X  -160.000, Y  +394.628, Z    +0.000, E1    -5.657, E3 +66170.159}
SPL {X  -160.000, Y  +401.354, Z    +0.000, E1   -13.067, E3 +66171.550}
SPL {X  -160.000, Y  +413.710, Z    +0.000, E1   -25.976, E3 +66176.342}
SPL {X  -160.000, Y  +449.556, Z    +0.000, E1   -44.518, E3 +66202.384}
SPL {X  -160.000, Y  +494.814, Z    +0.000, E1   -49.280, E3 +66260.733}
SPL {X  -160.000, Y  +504.699, Z    +0.000, E1   -49.282, E3 +66278.813}
SPL {X  -160.000, Y  +515.266, Z    +0.000, E1   -49.291, E3 +66298.127}
SPL {X  -160.000, Y  +526.314, Z    +0.000, E1   -49.296, E3 +66318.356}
SPL {X  -160.000, Y  +536.842, Z    +0.000, E1   -49.263, E3 +66337.682}
SPL {X  -160.000, Y  +547.071, Z    +0.000, E1   -49.286, E3 +66356.359}
SPL {X  -160.000, Y  +558.279, Z    +0.000, E1   -49.288, E3 +66376.863}
SPL {X  -160.000, Y  +568.309, Z    +0.000, E1   -49.259, E3 +66395.258}
SPL {X  -160.000, Y  +579.695, Z    +0.000, E1   -49.320, E3 +66415.988}
SPL {X  -160.000, Y  +592.166, Z    +0.000, E1   -49.294, E3 +66438.848}
SPL {X  -160.000, Y  +603.260, Z    +0.000, E1   -49.285, E3 +66459.173}
SPL {X  -160.000, Y  +615.079, Z    +0.000, E1   -49.301, E3 +66480.785}
SPL {X  -160.000, Y  +627.012, Z    +0.000, E1   -49.289, E3 +66502.637}
SPL {X  -160.000, Y  +638.544, Z    +0.000, E1   -49.285, E3 +66523.748}
SPL {X  -160.000, Y  +649.673, Z    +0.000, E1   -49.278, E3 +66544.121}
SPL {X  -160.000, Y  +661.315, Z    +0.000, E1   -49.297, E3 +66565.391}
SPL {X  -159.993, Y  +672.984, Z    +0.000, E1   -49.282, E3 +66586.782}
SPL {X  -159.528, Y  +683.783, Z    +0.000, E1   -49.201, E3 +66607.036}
SPL {X  -158.288, Y  +694.841, Z    +0.000, E1   -49.005, E3 +66628.550}
SPL {X  -156.479, Y  +704.881, Z    +0.000, E1   -48.644, E3 +66648.864}
SPL {X  -154.000, Y  +714.904, Z    +0.000, E1   -48.243, E3 +66669.673}
SPL {X  -150.967, Y  +724.498, Z    +0.000, E1   -47.642, E3 +66690.338}
SPL {X  -147.384, Y  +733.774, Z    +0.000, E1   -47.000, E3 +66710.811}
SPL {X  -139.301, Y  +750.209, Z    +0.000, E1   -41.935, E3 +66781.992}
ENDSPLINE

SPLINE
SPL {X  -151.875, Y  +721.838, Z    +0.000, E1   -27.241, E3 +66859.162}
SPL {X  -157.803, Y  +697.921, Z    +0.000, E1   -15.861, E3 +66875.029}
SPL {X  -159.710, Y  +681.128, Z    +0.000, E1    -6.465, E3 +66880.163}
SPL {X  -159.999, Y  +671.996, Z    +0.000, E1    -0.411, E3 +66881.493}
SPL {X  -160.000, Y  +665.132, Z    +0.000, E1    +5.902, E3 +66882.303}
SPL {X  -160.000, Y  +655.952, Z    +0.000, E1   +16.601, E3 +66884.299}
SPL {X  -160.000, Y  +643.612, Z    +0.000, E1   +29.091, E3 +66889.270}
SPL {X  -160.000, Y  +606.346, Z    +0.000, E1   +46.235, E3 +66917.078}
SPL {X  -160.000, Y  +564.751, Z    +0.000, E1   +49.682, E3 +66972.249}
SPL {X  -160.000, Y  +555.844, Z    +0.000, E1   +49.673, E3 +66988.330}
SPL {X  -160.000, Y  +545.889, Z    +0.000, E1   +49.702, E3 +67006.229}
SPL {X  -160.000, Y  +535.482, Z    +0.000, E1   +49.684, E3 +67025.028}
SPL {X  -160.000, Y  +526.440, Z    +0.000, E1   +49.666, E3 +67041.362}
SPL {X  -160.000, Y  +518.889, Z    +0.000, E1   +49.624, E3 +67055.186}
ENDSPLINE

SPLINE
SPL {X  -160.000, Y  +548.948, Z    +0.000, E1   +36.551, E3 +67064.875}
ENDSPLINE

SPLINE
SPL {X  -160.000, Y  +541.880, Z    +0.000, E1   +37.562, E3 +67078.653}
SPL {X  -160.000, Y  +532.200, Z    +0.000, E1   +38.842, E3 +67096.994}
SPL {X  -160.000, Y  +523.085, Z    +0.000, E1   +39.970, E3 +67113.685}
SPL {X  -160.000, Y  +513.603, Z    +0.000, E1   +41.139, E3 +67130.269}
SPL {X  -160.000, Y  +503.235, Z    +0.000, E1   +42.462, E3 +67146.977}
SPL {X  -160.000, Y  +493.516, Z    +0.000, E1   +43.493, E3 +67163.022}
SPL {X  -160.000, Y  +483.478, Z    +0.000, E1   +44.599, E3 +67178.480}
SPL {X  -160.000, Y  +473.020, Z    +0.000, E1   +45.665, E3 +67194.310}
SPL {X  -160.000, Y  +461.024, Z    +0.000, E1   +46.836, E3 +67211.785}
SPL {X  -160.000, Y  +448.988, Z    +0.000, E1   +48.043, E3 +67228.047}
SPL {X  -160.000, Y  +439.029, Z    +0.000, E1   +48.623, E3 +67243.454}
SPL {X  -160.000, Y  +429.710, Z    +0.000, E1   +48.622, E3 +67260.901}
SPL {X  -160.000, Y  +420.891, Z    +0.000, E1   +48.613, E3 +67277.426}
SPL {X  -160.000, Y  +412.565, Z    +0.000, E1   +48.611, E3 +67292.992}
SPL {X  -160.000, Y  +404.943, Z    +0.000, E1   +48.601, E3 +67307.294}
SPL {X  -160.000, Y  +395.837, Z    +0.000, E1   +48.634, E3 +67324.284}
SPL {X  -159.987, Y  +386.768, Z    +0.000, E1   +48.609, E3 +67341.288}
SPL {X  -159.620, Y  +377.782, Z    +0.000, E1   +48.569, E3 +67358.456}
SPL {X  -158.761, Y  +368.924, Z    +0.000, E1   +48.401, E3 +67375.983}
SPL {X  -157.560, Y  +360.964, Z    +0.000, E1   +48.177, E3 +67392.154}
SPL {X  -156.187, Y  +354.076, Z    +0.000, E1   +47.920, E3 +67406.487}
SPL {X  -154.507, Y  +347.236, Z    +0.000, E1   +47.623, E3 +67421.015}
SPL {X  -152.108, Y  +339.169, Z    +0.000, E1   +47.215, E3 +67438.492}
SPL {X  -149.264, Y  +331.177, Z    +0.000, E1   +46.657, E3 +67456.291}
SPL {X  -146.675, Y  +324.875, Z    +0.000, E1   +46.130, E3 +67470.644}
SPL {X  -140.793, Y  +312.792, Z    +0.000, E1   +40.077, E3 +67544.887}
ENDSPLINE

SPLINE
SPL {X  -154.674, Y  +347.860, Z    +0.000, E1   +23.016, E3 +67615.030}
SPL {X  -159.179, Y  +372.617, Z    +0.000, E1   +10.186, E3 +67627.679}
SPL {X  -159.924, Y  +383.861, Z    +0.000, E1    +3.320, E3 +67630.301}
SPL {X  -160.000, Y  +389.631, Z    +0.000, E1    -0.873, E3 +67631.017}
SPL {X  -160.000, Y  +394.628, Z    +0.000, E1    -5.657, E3 +67631.693}
SPL {X  -160.000, Y  +401.354, Z    +0.000, E1   -13.067, E3 +67633.084}
SPL {X  -160.000, Y  +413.710, Z    +0.000, E1   -25.976, E3 +67637.876}
SPL {X  -160.000, Y  +449.556, Z    +0.000, E1   -44.518, E3 +67663.918}
SPL {X  -160.000, Y  +494.814, Z    +0.000, E1   -49.280, E3 +67722.268}
SPL {X  -160.000, Y  +504.699, Z    +0.000, E1   -49.282, E3 +67740.347}
SPL {X  -160.000, Y  +515.266, Z    +0.000, E1   -49.291, E3 +67759.661}
SPL {X  -160.000, Y  +526.314, Z    +0.000, E1   -49.296, E3 +67779.890}
SPL {X  -160.000, Y  +536.842, Z    +0.000, E1   -49.263, E3 +67799.216}
SPL {X  -160.000, Y  +547.071, Z    +0.000, E1   -49.286, E3 +67817.893}
SPL {X  -160.000, Y  +558.279, Z    +0.000, E1   -49.288, E3 +67838.397}
SPL {X  -160.000, Y  +568.309, Z    +0.000, E1   -49.259, E3 +67856.792}
SPL {X  -160.000, Y  +579.695, Z    +0.000, E1   -49.320, E3 +67877.523}
SPL {X  -160.000, Y  +592.166, Z    +0.000, E1   -49.294, E3 +67900.382}
SPL {X  -160.000, Y  +603.260, Z    +0.000, E1   -49.285, E3 +67920.707}
SPL {X  -160.000, Y  +615.079, Z    +0.000, E1   -49.301, E3 +67942.319}
SPL {X  -160.000, Y  +627.012, Z    +0.000, E1   -49.289, E3 +67964.171}
SPL {X  -160.000, Y  +638.544, Z    +0.000, E1   -49.285, E3 +67985.282}
SPL {X  -160.000, Y  +649.673, Z    +0.000, E1   -49.278, E3 +68005.655}
SPL {X  -160.000, Y  +661.315, Z    +0.000, E1   -49.297, E3 +68026.925}
SPL {X  -159.993, Y  +672.984, Z    +0.000, E1   -49.282, E3 +68048.316}
SPL {X  -159.528, Y  +683.783, Z    +0.000, E1   -49.201, E3 +68068.570}
SPL {X  -158.288, Y  +694.841, Z    +0.000, E1   -49.005, E3 +68090.084}
SPL {X  -156.479, Y  +704.881, Z    +0.000, E1   -48.644, E3 +68110.398}
SPL {X  -154.000, Y  +714.904, Z    +0.000, E1   -48.243, E3 +68131.207}
SPL {X  -150.967, Y  +724.498, Z    +0.000, E1   -47.642, E3 +68151.872}
SPL {X  -147.384, Y  +733.774, Z    +0.000, E1   -47.000, E3 +68172.345}
SPL {X  -139.301, Y  +750.209, Z    +0.000, E1   -41.935, E3 +68243.526}
ENDSPLINE

SPLINE
SPL {X  -151.875, Y  +721.838, Z    +0.000, E1   -27.241, E3 +68320.697}
SPL {X  -157.803, Y  +697.921, Z    +0.000, E1   -15.861, E3 +68336.564}
SPL {X  -159.710, Y  +681.128, Z    +0.000, E1    -6.465, E3 +68341.697}
SPL {X  -159.999, Y  +671.996, Z    +0.000, E1    -0.411, E3 +68343.027}
SPL {X  -160.000, Y  +665.132, Z    +0.000, E1    +5.902, E3 +68343.837}
SPL {X  -160.000, Y  +655.952, Z    +0.000, E1   +16.601, E3 +68345.833}
SPL {X  -160.000, Y  +643.612, Z    +0.000, E1   +29.091, E3 +68350.804}
SPL {X  -160.000, Y  +606.346, Z    +0.000, E1   +46.235, E3 +68378.612}
SPL {X  -160.000, Y  +564.751, Z    +0.000, E1   +49.682, E3 +68433.784}
SPL {X  -160.000, Y  +555.844, Z    +0.000, E1   +49.673, E3 +68449.864}
SPL {X  -160.000, Y  +545.889, Z    +0.000, E1   +49.702, E3 +68467.763}
SPL {X  -160.000, Y  +535.482, Z    +0.000, E1   +49.684, E3 +68486.563}
SPL {X  -160.000, Y  +526.440, Z    +0.000, E1   +49.666, E3 +68502.896}
SPL {X  -160.000, Y  +518.889, Z    +0.000, E1   +49.624, E3 +68516.720}
ENDSPLINE

SPLINE
SPL {X  -160.000, Y  +548.948, Z    +0.000, E1   +36.551, E3 +68526.409}
ENDSPLINE

SPLINE
SPL {X  -160.000, Y  +541.880, Z    +0.000, E1   +37.562, E3 +68540.187}
SPL {X  -160.000, Y  +532.200, Z    +0.000, E1   +38.842, E3 +68558.528}
SPL {X  -160.000, Y  +523.085, Z    +0.000, E1   +39.970, E3 +68575.219}
SPL {X  -160.000, Y  +513.603, Z    +0.000, E1   +41.139, E3 +68591.803}
SPL {X  -160.000, Y  +503.235, Z    +0.000, E1   +42.462, E3 +68608.511}
SPL {X  -160.000, Y  +493.516, Z    +0.000, E1   +43.493, E3 +68624.556}
SPL {X  -160.000, Y  +483.478, Z    +0.000, E1   +44.599, E3 +68640.014}
SPL {X  -160.000, Y  +473.020, Z    +0.000, E1   +45.665, E3 +68655.844}
SPL {X  -160.000, Y  +461.024, Z    +0.000, E1   +46.836, E3 +68673.319}
SPL {X  -160.000, Y  +448.988, Z    +0.000, E1   +48.043, E3 +68689.581}
SPL {X  -160.000, Y  +439.029, Z    +0.000, E1   +48.623, E3 +68704.988}
SPL {X  -160.000, Y  +429.710, Z    +0.000, E1   +48.622, E3 +68722.435}
SPL {X  -160.000, Y  +420.891, Z    +0.000, E1   +48.613, E3 +68738.960}
SPL {X  -160.000, Y  +412.565, Z    +0.000, E1   +48.611, E3 +68754.526}
SPL {X  -160.000, Y  +404.943, Z    +0.000, E1   +48.601, E3 +68768.828}
SPL {X  -160.000, Y  +395.837, Z    +0.000, E1   +48.634, E3 +68785.818}
SPL {X  -159.987, Y  +386.768, Z    +0.000, E1   +48.609, E3 +68802.822}
SPL {X  -159.620, Y  +377.782, Z    +0.000, E1   +48.569, E3 +68819.990}
SPL {X  -158.761, Y  +368.924, Z    +0.000, E1   +48.401, E3 +68837.517}
SPL {X  -157.560, Y  +360.964, Z    +0.000, E1   +48.177, E3 +68853.688}
SPL {X  -156.187, Y  +354.076, Z    +0.000, E1   +47.920, E3 +68868.021}
SPL {X  -154.507, Y  +347.236, Z    +0.000, E1   +47.623, E3 +68882.549}
SPL {X  -152.108, Y  +339.169, Z    +0.000, E1   +47.215, E3 +68900.027}
SPL {X  -149.264, Y  +331.177, Z    +0.000, E1   +46.657, E3 +68917.825}
SPL {X  -146.675, Y  +324.875, Z    +0.000, E1   +46.130, E3 +68932.178}
SPL {X  -140.793, Y  +312.792, Z    +0.000, E1   +40.077, E3 +69006.422}
ENDSPLINE

SPLINE
SPL {X  -154.674, Y  +347.860, Z    +0.000, E1   +23.016, E3 +69076.565}
SPL {X  -159.179, Y  +372.617, Z    +0.000, E1   +10.186, E3 +69089.213}
SPL {X  -159.924, Y  +383.861, Z    +0.000, E1    +3.320, E3 +69091.836}
SPL {X  -160.000, Y  +389.631, Z    +0.000, E1    -0.873, E3 +69092.551}
SPL {X  -160.000, Y  +394.628, Z    +0.000, E1    -5.657, E3 +69093.227}
SPL {X  -160.000, Y  +401.354, Z    +0.000, E1   -13.067, E3 +69094.618}
SPL {X  -160.000, Y  +413.710, Z    +0.000, E1   -25.976, E3 +69099.411}
SPL {X  -160.000, Y  +449.556, Z    +0.000, E1   -44.518, E3 +69125.452}
SPL {X  -160.000, Y  +494.814, Z    +0.000, E1   -49.280, E3 +69183.802}
SPL {X  -160.000, Y  +504.699, Z    +0.000, E1   -49.282, E3 +69201.881}
SPL {X  -160.000, Y  +515.266, Z    +0.000, E1   -49.291, E3 +69221.195}
SPL {X  -160.000, Y  +526.314, Z    +0.000, E1   -49.296, E3 +69241.424}
SPL {X  -160.000, Y  +536.842, Z    +0.000, E1   -49.263, E3 +69260.750}
SPL {X  -160.000, Y  +547.071, Z    +0.000, E1   -49.286, E3 +69279.427}
SPL {X  -160.000, Y  +558.279, Z    +0.000, E1   -49.288, E3 +69299.931}
SPL {X  -160.000, Y  +568.309, Z    +0.000, E1   -49.259, E3 +69318.326}
SPL {X  -160.000, Y  +579.695, Z    +0.000, E1   -49.320, E3 +69339.057}
SPL {X  -160.000, Y  +592.166, Z    +0.000, E1   -49.294, E3 +69361.916}
SPL {X  -160.000, Y  +603.260, Z    +0.000, E1   -49.285, E3 +69382.241}
SPL {X  -160.000, Y  +615.079, Z    +0.000, E1   -49.301, E3 +69403.853}
SPL {X  -160.000, Y  +627.012, Z    +0.000, E1   -49.289, E3 +69425.706}
SPL {X  -160.000, Y  +638.544, Z    +0.000, E1   -49.285, E3 +69446.816}
SPL {X  -160.000, Y  +649.673, Z    +0.000, E1   -49.278, E3 +69467.189}
SPL {X  -160.000, Y  +661.315, Z    +0.000, E1   -49.297, E3 +69488.459}
SPL {X  -159.993, Y  +672.984, Z    +0.000, E1   -49.282, E3 +69509.850}
SPL {X  -159.528, Y  +683.783, Z    +0.000, E1   -49.201, E3 +69530.105}
SPL {X  -158.288, Y  +694.841, Z    +0.000, E1   -49.005, E3 +69551.618}
SPL {X  -156.479, Y  +704.881, Z    +0.000, E1   -48.644, E3 +69571.932}
SPL {X  -154.000, Y  +714.904, Z    +0.000, E1   -48.243, E3 +69592.741}
SPL {X  -150.967, Y  +724.498, Z    +0.000, E1   -47.642, E3 +69613.407}
SPL {X  -147.384, Y  +733.774, Z    +0.000, E1   -47.000, E3 +69633.879}
SPL {X  -139.301, Y  +750.209, Z    +0.000, E1   -41.935, E3 +69705.060}
ENDSPLINE

SPLINE
SPL {X  -151.875, Y  +721.838, Z    +0.000, E1   -27.241, E3 +69782.231}
SPL {X  -157.803, Y  +697.921, Z    +0.000, E1   -15.861, E3 +69798.098}
SPL {X  -159.710, Y  +681.128, Z    +0.000, E1    -6.465, E3 +69803.231}
SPL {X  -159.999, Y  +671.996, Z    +0.000, E1    -0.411, E3 +69804.561}
SPL {X  -160.000, Y  +665.132, Z    +0.000, E1    +5.902, E3 +69805.372}
SPL {X  -160.000, Y  +655.952, Z    +0.000, E1   +16.601, E3 +69807.367}
SPL {X  -160.000, Y  +643.612, Z    +0.000, E1   +29.091, E3 +69812.338}
SPL {X  -160.000, Y  +606.346, Z    +0.000, E1   +46.235, E3 +69840.146}
SPL {X  -160.000, Y  +564.751, Z    +0.000, E1   +49.682, E3 +69895.318}
SPL {X  -160.000, Y  +555.844, Z    +0.000, E1   +49.673, E3 +69911.398}
SPL {X  -160.000, Y  +545.889, Z    +0.000, E1   +49.702, E3 +69929.297}
SPL {X  -160.000, Y  +535.482, Z    +0.000, E1   +49.684, E3 +69948.097}
SPL {X  -160.000, Y  +526.440, Z    +0.000, E1   +49.666, E3 +69964.430}
SPL {X  -160.000, Y  +518.889, Z    +0.000, E1   +49.624, E3 +69978.254}
ENDSPLINE

SPLINE
SPL {X  -160.000, Y  +548.948, Z    +0.000, E1   +36.551, E3 +69987.943}
ENDSPLINE

SPLINE
SPL {X  -160.000, Y  +541.880, Z    +0.000, E1   +37.562, E3 +70001.721}
SPL {X  -160.000, Y  +532.200, Z    +0.000, E1   +38.842, E3 +70020.063}
SPL {X  -160.000, Y  +523.085, Z    +0.000, E1   +39.970, E3 +70036.753}
SPL {X  -160.000, Y  +513.603, Z    +0.000, E1   +41.139, E3 +70053.337}
SPL {X  -160.000, Y  +503.235, Z    +0.000, E1   +42.462, E3 +70070.045}
SPL {X  -160.000, Y  +493.516, Z    +0.000, E1   +43.493, E3 +70086.090}
SPL {X  -160.000, Y  +483.478, Z    +0.000, E1   +44.599, E3 +70101.548}
SPL {X  -160.000, Y  +473.020, Z    +0.000, E1   +45.665, E3 +70117.378}
SPL {X  -160.000, Y  +461.024, Z    +0.000, E1   +46.836, E3 +70134.853}
SPL {X  -160.000, Y  +448.988, Z    +0.000, E1   +48.043, E3 +70151.115}
SPL {X  -160.000, Y  +439.029, Z    +0.000, E1   +48.623, E3 +70166.523}
SPL {X  -160.000, Y  +429.710, Z    +0.000, E1   +48.622, E3 +70183.969}
SPL {X  -160.000, Y  +420.891, Z    +0.000, E1   +48.613, E3 +70200.494}
SPL {X  -160.000, Y  +412.565, Z    +0.000, E1   +48.611, E3 +70216.060}
SPL {X  -160.000, Y  +404.943, Z    +0.000, E1   +48.601, E3 +70230.362}
SPL {X  -160.000, Y  +395.837, Z    +0.000, E1   +48.634, E3 +70247.352}
SPL {X  -159.987, Y  +386.768, Z    +0.000, E1   +48.609, E3 +70264.356}
SPL {X  -159.620, Y  +377.782, Z    +0.000, E1   +48.569, E3 +70281.524}
SPL {X  -158.761, Y  +368.924, Z    +0.000, E1   +48.401, E3 +70299.051}
SPL {X  -157.560, Y  +360.964, Z    +0.000, E1   +48.177, E3 +70315.223}
SPL {X  -156.187, Y  +354.076, Z    +0.000, E1   +47.920, E3 +70329.555}
SPL {X  -154.507, Y  +347.236, Z    +0.000, E1   +47.623, E3 +70344.083}
SPL {X  -152.108, Y  +339.169, Z    +0.000, E1   +47.215, E3 +70361.561}
SPL {X  -149.264, Y  +331.177, Z    +0.000, E1   +46.657, E3 +70379.360}
SPL {X  -146.675, Y  +324.875, Z    +0.000, E1   +46.130, E3 +70393.712}
SPL {X  -140.793, Y  +312.792, Z    +0.000, E1   +40.077, E3 +70467.956}
ENDSPLINE

SPLINE
SPL {X  -154.674, Y  +347.860, Z    +0.000, E1   +23.016, E3 +70538.099}
SPL {X  -159.179, Y  +372.617, Z    +0.000, E1   +10.186, E3 +70550.747}
SPL {X  -159.924, Y  +383.861, Z    +0.000, E1    +3.320, E3 +70553.370}
SPL {X  -160.000, Y  +389.631, Z    +0.000, E1    -0.873, E3 +70554.085}
SPL {X  -160.000, Y  +394.628, Z    +0.000, E1    -5.657, E3 +70554.761}
SPL {X  -160.000, Y  +401.354, Z    +0.000, E1   -13.067, E3 +70556.152}
SPL {X  -160.000, Y  +413.710, Z    +0.000, E1   -25.976, E3 +70560.945}
SPL {X  -160.000, Y  +449.556, Z    +0.000, E1   -44.518, E3 +70586.986}
SPL {X  -160.000, Y  +494.814, Z    +0.000, E1   -49.280, E3 +70645.336}
SPL {X  -160.000, Y  +504.699, Z    +0.000, E1   -49.282, E3 +70663.416}
SPL {X  -160.000, Y  +515.266, Z    +0.000, E1   -49.291, E3 +70682.729}
SPL {X  -160.000, Y  +526.314, Z    +0.000, E1   -49.296, E3 +70702.959}
SPL {X  -160.000, Y  +536.842, Z    +0.000, E1   -49.263, E3 +70722.285}
SPL {X  -160.000, Y  +547.071, Z    +0.000, E1   -49.286, E3 +70740.961}
SPL {X  -160.000, Y  +558.279, Z    +0.000, E1   -49.288, E3 +70761.465}
SPL {X  -160.000, Y  +568.309, Z    +0.000, E1   -49.259, E3 +70779.860}
SPL {X  -160.000, Y  +579.695, Z    +0.000, E1   -49.320, E3 +70800.591}
SPL {X  -160.000, Y  +592.166, Z    +0.000, E1   -49.294, E3 +70823.451}
SPL {X  -160.000, Y  +603.260, Z    +0.000, E1   -49.285, E3 +70843.775}
SPL {X  -160.000, Y  +615.079, Z    +0.000, E1   -49.301, E3 +70865.387}
SPL {X  -160.000, Y  +627.012, Z    +0.000, E1   -49.289, E3 +70887.240}
SPL {X  -160.000, Y  +638.544, Z    +0.000, E1   -49.285, E3 +70908.350}
SPL {X  -160.000, Y  +649.673, Z    +0.000, E1   -49.278, E3 +70928.723}
SPL {X  -160.000, Y  +661.315, Z    +0.000, E1   -49.297, E3 +70949.994}
SPL {X  -159.993, Y  +672.984, Z    +0.000, E1   -49.282, E3 +70971.384}
SPL {X  -159.528, Y  +683.783, Z    +0.000, E1   -49.201, E3 +70991.639}
SPL {X  -158.288, Y  +694.841, Z    +0.000, E1   -49.005, E3 +71013.152}
SPL {X  -156.479, Y  +704.881, Z    +0.000, E1   -48.644, E3 +71033.466}
SPL {X  -154.000, Y  +714.904, Z    +0.000, E1   -48.243, E3 +71054.275}
SPL {X  -150.967, Y  +724.498, Z    +0.000, E1   -47.642, E3 +71074.941}
SPL {X  -147.384, Y  +733.774, Z    +0.000, E1   -47.000, E3 +71095.414}
SPL {X  -139.301, Y  +750.209, Z    +0.000, E1   -41.935, E3 +71166.594}
ENDSPLINE

SPLINE
SPL {X  -151.875, Y  +721.838, Z    +0.000, E1   -27.241, E3 +71243.765}
SPL {X  -157.803, Y  +697.921, Z    +0.000, E1   -15.861, E3 +71259.632}
SPL {X  -159.710, Y  +681.128, Z    +0.000, E1    -6.465, E3 +71264.765}
SPL {X  -159.999, Y  +671.996, Z    +0.000, E1    -0.411, E3 +71266.096}
SPL {X  -160.000, Y  +665.132, Z    +0.000, E1    +5.902, E3 +71266.906}
SPL {X  -160.000, Y  +655.952, Z    +0.000, E1   +16.601, E3 +71268.901}
SPL {X  -160.000, Y  +643.612, Z    +0.000, E1   +29.091, E3 +71273.872}
SPL {X  -160.000, Y  +606.346, Z    +0.000, E1   +46.235, E3 +71301.680}
SPL {X  -160.000, Y  +564.751, Z    +0.000, E1   +49.682, E3 +71356.852}
SPL {X  -160.000, Y  +555.844, Z    +0.000, E1   +49.673, E3 +71372.933}
SPL {X  -160.000, Y  +545.889, Z    +0.000, E1   +49.702, E3 +71390.831}
SPL {X  -160.000, Y  +535.482, Z    +0.000, E1   +49.684, E3 +71409.631}
SPL {X  -160.000, Y  +526.440, Z    +0.000, E1   +49.666, E3 +71425.964}
SPL {X  -160.000, Y  +518.889, Z    +0.000, E1   +49.624, E3 +71439.788}
ENDSPLINE

SPLINE
SPL {X  -160.000, Y  +548.948, Z    +0.000, E1   +36.551, E3 +71449.477}
ENDSPLINE

SPLINE
SPL {X  -160.000, Y  +541.880, Z    +0.000, E1   +37.562, E3 +71463.255}
SPL {X  -160.000, Y  +532.200, Z    +0.000, E1   +38.842, E3 +71481.597}
SPL {X  -160.000, Y  +523.085, Z    +0.000, E1   +39.970, E3 +71498.287}
SPL {X  -160.000, Y  +513.603, Z    +0.000, E1   +41.139, E3 +71514.871}
SPL {X  -160.000, Y  +503.235, Z    +0.000, E1   +42.462, E3 +71531.579}
SPL {X  -160.000, Y  +493.516, Z    +0.000, E1   +43.493, E3 +71547.624}
SPL {X  -160.000, Y  +483.478, Z    +0.000, E1   +44.599, E3 +71563.082}
SPL {X  -160.000, Y  +473.020, Z    +0.000, E1   +45.665, E3 +71578.912}
SPL {X  -160.000, Y  +461.024, Z    +0.000, E1   +46.836, E3 +71596.387}
SPL {X  -160.000, Y  +448.988, Z    +0.000, E1   +48.043, E3 +71612.649}
ENDSPLINE

SPLINE
SPL {X  -160.000, Y  +451.951, Z    +0.000, E1   +44.355, E3 +71628.699}
SPL {X  -160.000, Y  +442.331, Z    +0.000, E1   +44.390, E3 +71649.563}
SPL {X  -160.000, Y  +433.037, Z    +0.000, E1   +44.348, E3 +71669.837}
SPL {X  -160.000, Y  +424.435, Z    +0.000, E1   +44.358, E3 +71688.506}
SPL {X  -160.000, Y  +416.015, Z    +0.000, E1   +44.348, E3 +71706.826}
SPL {X  -160.000, Y  +407.167, Z    +0.000, E1   +44.365, E3 +71726.036}
SPL {X  -160.000, Y  +397.599, Z    +0.000, E1   +44.371, E3 +71746.845}
SPL {X  -160.000, Y  +388.533, Z    +0.000, E1   +44.340, E3 +71766.620}
SPL {X  -159.759, Y  +380.021, Z    +0.000, E1   +44.311, E3 +71785.352}
SPL {X  -159.014, Y  +371.065, Z    +0.000, E1   +44.193, E3 +71805.590}
SPL {X  -157.745, Y  +362.030, Z    +0.000, E1   +43.965, E3 +71826.572}
SPL {X  -156.258, Y  +354.400, Z    +0.000, E1   +43.653, E3 +71844.779}
SPL {X  -154.385, Y  +346.786, Z    +0.000, E1   +43.356, E3 +71863.191}
SPL {X  -152.146, Y  +339.286, Z    +0.000, E1   +42.904, E3 +71881.825}
SPL {X  -149.854, Y  +332.731, Z    +0.000, E1   +42.474, E3 +71898.353}
SPL {X  -145.635, Y  +322.541, Z    +0.000, E1   +36.397, E3 +71974.312}
ENDSPLINE

SPLINE
SPL {X  -156.682, Y  +356.385, Z    +0.000, E1   +19.033, E3 +72032.618}
SPL {X  -159.526, Y  +376.492, Z    +0.000, E1    +8.067, E3 +72042.527}
SPL {X  -159.961, Y  +385.275, Z    +0.000, E1    +2.550, E3 +72044.566}
SPL {X  -160.000, Y  +390.345, Z    +0.000, E1    -1.188, E3 +72045.292}
SPL {X  -160.000, Y  +395.838, Z    +0.000, E1    -6.211, E3 +72046.235}
SPL {X  -160.000, Y  +403.277, Z    +0.000, E1   -14.057, E3 +72048.186}
SPL {X  -160.000, Y  +414.316, Z    +0.000, E1   -24.810, E3 +72053.259}
SPL {X  -160.000, Y  +442.604, Z    +0.000, E1   -40.161, E3 +72075.394}
SPL {X  -160.000, Y  +482.867, Z    +0.000, E1   -45.148, E3 +72135.610}
SPL {X  -160.000, Y  +494.769, Z    +0.000, E1   -45.151, E3 +72160.829}
SPL {X  -160.000, Y  +505.761, Z    +0.000, E1   -45.118, E3 +72184.143}
SPL {X  -160.000, Y  +517.347, Z    +0.000, E1   -45.173, E3 +72208.581}
SPL {X  -160.000, Y  +529.298, Z    +0.000, E1   -45.138, E3 +72233.964}
SPL {X  -160.000, Y  +540.664, Z    +0.000, E1   -45.139, E3 +72258.042}
SPL {X  -160.000, Y  +552.011, Z    +0.000, E1   -45.139, E3 +72282.078}
SPL {X  -160.000, Y  +563.667, Z    +0.000, E1   -45.146, E3 +72306.758}
SPL {X  -160.000, Y  +574.965, Z    +0.000, E1   -45.125, E3 +72330.734}
SPL {X  -160.000, Y  +585.644, Z    +0.000, E1   -45.117, E3 +72353.374}
SPL {X  -160.000, Y  +596.819, Z    +0.000, E1   -45.144, E3 +72377.015}
SPL {X  -160.000, Y  +608.165, Z    +0.000, E1   -45.120, E3 +72401.090}
SPL {X  -160.000, Y  +619.270, Z    +0.000, E1   -45.132, E3 +72424.592}
SPL {X  -160.000, Y  +629.968, Z    +0.000, E1   -45.117, E3 +72447.258}
SPL {X  -160.000, Y  +640.750, Z    +0.000, E1   -45.131, E3 +72470.081}
SPL {X  -160.000, Y  +651.429, Z    +0.000, E1   -45.117, E3 +72492.723}
SPL {X  -160.000, Y  +662.434, Z    +0.000, E1   -45.129, E3 +72516.067}
SPL {X  -159.992, Y  +673.110, Z    +0.000, E1   -45.097, E3 +72538.759}
SPL {X  -159.521, Y  +683.874, Z    +0.000, E1   -45.054, E3 +72562.015}
SPL {X  -158.435, Y  +693.823, Z    +0.000, E1   -44.810, E3 +72584.319}
SPL {X  -156.807, Y  +703.304, Z    +0.000, E1   -44.558, E3 +72606.039}
SPL {X  -154.802, Y  +711.950, Z    +0.000, E1   -44.141, E3 +72626.499}
SPL {X  -152.641, Y  +719.464, Z    +0.000, E1   -43.749, E3 +72644.615}
SPL {X  -149.826, Y  +727.645, Z    +0.000, E1   -43.252, E3 +72664.718}
SPL {X  -145.307, Y  +738.478, Z    +0.000, E1   -36.676, E3 +72744.786}
ENDSPLINE

SPLINE
SPL {X  -155.601, Y  +708.762, Z    +0.000, E1   -21.463, E3 +72799.572}
SPL {X  -158.549, Y  +693.002, Z    +0.000, E1   -13.406, E3 +72808.563}
SPL {X  -159.716, Y  +681.031, Z    +0.000, E1    -6.529, E3 +72812.713}
SPL {X  -160.000, Y  +671.641, Z    +0.000, E1    -0.547, E3 +72814.430}
SPL {X  -160.000, Y  +665.424, Z    +0.000, E1    +5.044, E3 +72815.378}
SPL {X  -160.000, Y  +658.015, Z    +0.000, E1   +12.630, E3 +72817.296}
SPL {X  -160.000, Y  +645.110, Z    +0.000, E1   +25.142, E3 +72823.096}
SPL {X  -160.000, Y  +611.664, Z    +0.000, E1   +41.262, E3 +72852.825}
SPL {X  -160.000, Y  +581.433, Z    +0.000, E1   +44.103, E3 +72902.562}
SPL {X  -160.000, Y  +572.090, Z    +0.000, E1   +44.120, E3 +72923.027}
SPL {X  -160.000, Y  +563.431, Z    +0.000, E1   +44.084, E3 +72942.080}
SPL {X  -160.000, Y  +556.107, Z    +0.000, E1   +44.076, E3 +72958.148}
SPL {X  -160.000, Y  +549.181, Z    +0.000, E1   +44.079, E3 +72973.308}
SPL {X  -160.000, Y  +542.413, Z    +0.000, E1   +44.088, E3 +72988.142}
SPL {X  -160.000, Y  +534.609, Z    +0.000, E1   +44.095, E3 +73005.252}
SPL {X  -160.000, Y  +527.457, Z    +0.000, E1   +44.070, E3 +73020.962}
SPL {X  -160.000, Y  +520.912, Z    +0.000, E1   +44.079, E3 +73035.303}
SPL {X  -160.000, Y  +514.086, Z    +0.000, E1   +44.081, E3 +73050.251}
SPL {X  -160.000, Y  +507.208, Z    +0.000, E1   +44.082, E3 +73065.328}
SPL {X  -160.000, Y  +499.184, Z    +0.000, E1   +44.113, E3 +73082.886}
ENDSPLINE

SPLINE
SPL {X  -160.000, Y  +503.824, Z    +0.000, E1   +39.488, E3 +73098.934}
ENDSPLINE

SPLINE
SPL {X  -160.000, Y  +499.279, Z    +0.000, E1   +38.981, E3 +73113.924}
SPL {X  -160.000, Y  +490.068, Z    +0.000, E1   +40.198, E3 +73130.229}
SPL {X  -160.000, Y  +481.368, Z    +0.000, E1   +41.274, E3 +73145.218}
SPL {X  -160.000, Y  +470.910, Z    +0.000, E1   +42.658, E3 +73161.727}
SPL {X  -160.000, Y  +460.219, Z    +0.000, E1   +43.912, E3 +73178.348}
SPL {X  -160.000, Y  +451.951, Z    +0.000, E1   +44.355, E3 +73193.913}
SPL {X  -160.000, Y  +442.331, Z    +0.000, E1   +44.390, E3 +73214.777}
SPL {X  -160.000, Y  +433.037, Z    +0.000, E1   +44.348, E3 +73235.051}
SPL {X  -160.000, Y  +424.435, Z    +0.000, E1   +44.358, E3 +73253.720}
SPL {X  -160.000, Y  +416.015, Z    +0.000, E1   +44.348, E3 +73272.040}
SPL {X  -160.000, Y  +407.167, Z    +0.000, E1   +44.365, E3 +73291.251}
SPL {X  -160.000, Y  +397.599, Z    +0.000, E1   +44.371, E3 +73312.059}
SPL {X  -160.000, Y  +388.533, Z    +0.000, E1   +44.340, E3 +73331.834}
SPL {X  -159.759, Y  +380.021, Z    +0.000, E1   +44.311, E3 +73350.566}
SPL {X  -159.014, Y  +371.065, Z    +0.000, E1   +44.193, E3 +73370.804}
SPL {X  -157.745, Y  +362.030, Z    +0.000, E1   +43.965, E3 +73391.786}
SPL {X  -156.258, Y  +354.400, Z    +0.000, E1   +43.653, E3 +73409.993}
SPL {X  -154.385, Y  +346.786, Z    +0.000, E1   +43.356, E3 +73428.405}
SPL {X  -152.146, Y  +339.286, Z    +0.000, E1   +42.904, E3 +73447.040}
SPL {X  -149.854, Y  +332.731, Z    +0.000, E1   +42.474, E3 +73463.567}
SPL {X  -145.635, Y  +322.541, Z    +0.000, E1   +36.397, E3 +73539.526}
ENDSPLINE

SPLINE
SPL {X  -156.682, Y  +356.385, Z    +0.000, E1   +19.033, E3 +73597.832}
SPL {X  -159.526, Y  +376.492, Z    +0.000, E1    +8.067, E3 +73607.741}
SPL {X  -159.961, Y  +385.275, Z    +0.000, E1    +2.550, E3 +73609.780}
SPL {X  -160.000, Y  +390.345, Z    +0.000, E1    -1.188, E3 +73610.506}
SPL {X  -160.000, Y  +395.838, Z    +0.000, E1    -6.211, E3 +73611.449}
SPL {X  -160.000, Y  +403.277, Z    +0.000, E1   -14.057, E3 +73613.401}
SPL {X  -160.000, Y  +414.316, Z    +0.000, E1   -24.810, E3 +73618.474}
SPL {X  -160.000, Y  +442.604, Z    +0.000, E1   -40.161, E3 +73640.608}
SPL {X  -160.000, Y  +482.867, Z    +0.000, E1   -45.148, E3 +73700.824}
SPL {X  -160.000, Y  +494.769, Z    +0.000, E1   -45.151, E3 +73726.043}
SPL {X  -160.000, Y  +505.761, Z    +0.000, E1   -45.118, E3 +73749.357}
SPL {X  -160.000, Y  +517.347, Z    +0.000, E1   -45.173, E3 +73773.795}
SPL {X  -160.000, Y  +529.298, Z    +0.000, E1   -45.138, E3 +73799.178}
SPL {X  -160.000, Y  +540.664, Z    +0.000, E1   -45.139, E3 +73823.256}
SPL {X  -160.000, Y  +552.011, Z    +0.000, E1   -45.139, E3 +73847.292}
SPL {X  -160.000, Y  +563.667, Z    +0.000, E1   -45.146, E3 +73871.972}
SPL {X  -160.000, Y  +574.965, Z    +0.000, E1   -45.125, E3 +73895.948}
SPL {X  -160.000, Y  +585.644, Z    +0.000, E1   -45.117, E3 +73918.588}
SPL {X  -160.000, Y  +596.819, Z    +0.000, E1   -45.144, E3 +73942.229}
SPL {X  -160.000, Y  +608.165, Z    +0.000, E1   -45.120, E3 +73966.304}
SPL {X  -160.000, Y  +619.270, Z    +0.000, E1   -45.132, E3 +73989.806}
SPL {X  -160.000, Y  +629.968, Z    +0.000, E1   -45.117, E3 +74012.473}
SPL {X  -160.000, Y  +640.750, Z    +0.000, E1   -45.131, E3 +74035.296}
SPL {X  -160.000, Y  +651.429, Z    +0.000, E1   -45.117, E3 +74057.937}
SPL {X  -160.000, Y  +662.434, Z    +0.000, E1   -45.129, E3 +74081.281}
SPL {X  -159.992, Y  +673.110, Z    +0.000, E1   -45.097, E3 +74103.974}
SPL {X  -159.521, Y  +683.874, Z    +0.000, E1   -45.054, E3 +74127.229}
SPL {X  -158.435, Y  +693.823, Z    +0.000, E1   -44.810, E3 +74149.533}
SPL {X  -156.807, Y  +703.304, Z    +0.000, E1   -44.558, E3 +74171.254}
SPL {X  -154.802, Y  +711.950, Z    +0.000, E1   -44.141, E3 +74191.714}
SPL {X  -152.641, Y  +719.464, Z    +0.000, E1   -43.749, E3 +74209.829}
SPL {X  -149.826, Y  +727.645, Z    +0.000, E1   -43.252, E3 +74229.932}
SPL {X  -145.307, Y  +738.478, Z    +0.000, E1   -36.676, E3 +74310.000}
ENDSPLINE

SPLINE
SPL {X  -155.601, Y  +708.762, Z    +0.000, E1   -21.463, E3 +74364.787}
SPL {X  -158.549, Y  +693.002, Z    +0.000, E1   -13.406, E3 +74373.777}
SPL {X  -159.716, Y  +681.031, Z    +0.000, E1    -6.529, E3 +74377.927}
SPL {X  -160.000, Y  +671.641, Z    +0.000, E1    -0.547, E3 +74379.644}
SPL {X  -160.000, Y  +665.424, Z    +0.000, E1    +5.044, E3 +74380.592}
SPL {X  -160.000, Y  +658.015, Z    +0.000, E1   +12.630, E3 +74382.510}
SPL {X  -160.000, Y  +645.110, Z    +0.000, E1   +25.142, E3 +74388.310}
SPL {X  -160.000, Y  +611.664, Z    +0.000, E1   +41.262, E3 +74418.040}
SPL {X  -160.000, Y  +581.433, Z    +0.000, E1   +44.103, E3 +74467.776}
SPL {X  -160.000, Y  +572.090, Z    +0.000, E1   +44.120, E3 +74488.241}
SPL {X  -160.000, Y  +563.431, Z    +0.000, E1   +44.084, E3 +74507.294}
SPL {X  -160.000, Y  +556.107, Z    +0.000, E1   +44.076, E3 +74523.362}
SPL {X  -160.000, Y  +549.181, Z    +0.000, E1   +44.079, E3 +74538.522}
SPL {X  -160.000, Y  +542.413, Z    +0.000, E1   +44.088, E3 +74553.356}
SPL {X  -160.000, Y  +534.609, Z    +0.000, E1   +44.095, E3 +74570.466}
SPL {X  -160.000, Y  +527.457, Z    +0.000, E1   +44.070, E3 +74586.176}
SPL {X  -160.000, Y  +520.912, Z    +0.000, E1   +44.079, E3 +74600.517}
SPL {X  -160.000, Y  +514.086, Z    +0.000, E1   +44.081, E3 +74615.465}
SPL {X  -160.000, Y  +507.208, Z    +0.000, E1   +44.082, E3 +74630.542}
SPL {X  -160.000, Y  +499.184, Z    +0.000, E1   +44.113, E3 +74648.100}
ENDSPLINE

SPLINE
SPL {X  -160.000, Y  +503.824, Z    +0.000, E1   +39.488, E3 +74664.149}
ENDSPLINE

SPLINE
SPL {X  -160.000, Y  +499.279, Z    +0.000, E1   +38.981, E3 +74679.139}
SPL {X  -160.000, Y  +490.068, Z    +0.000, E1   +40.198, E3 +74695.443}
SPL {X  -160.000, Y  +481.368, Z    +0.000, E1   +41.274, E3 +74710.433}
SPL {X  -160.000, Y  +470.910, Z    +0.000, E1   +42.658, E3 +74726.941}
SPL {X  -160.000, Y  +460.219, Z    +0.000, E1   +43.912, E3 +74743.562}
SPL {X  -160.000, Y  +451.951, Z    +0.000, E1   +44.355, E3 +74759.127}
SPL {X  -160.000, Y  +442.331, Z    +0.000, E1   +44.390, E3 +74779.991}
SPL {X  -160.000, Y  +433.037, Z    +0.000, E1   +44.348, E3 +74800.266}
SPL {X  -160.000, Y  +424.435, Z    +0.000, E1   +44.358, E3 +74818.934}
SPL {X  -160.000, Y  +416.015, Z    +0.000, E1   +44.348, E3 +74837.254}
SPL {X  -160.000, Y  +407.167, Z    +0.000, E1   +44.365, E3 +74856.465}
SPL {X  -160.000, Y  +397.599, Z    +0.000, E1   +44.371, E3 +74877.273}
SPL {X  -160.000, Y  +388.533, Z    +0.000, E1   +44.340, E3 +74897.048}
SPL {X  -159.759, Y  +380.021, Z    +0.000, E1   +44.311, E3 +74915.780}
SPL {X  -159.014, Y  +371.065, Z    +0.000, E1   +44.193, E3 +74936.018}
SPL {X  -157.745, Y  +362.030, Z    +0.000, E1   +43.965, E3 +74957.000}
SPL {X  -156.258, Y  +354.400, Z    +0.000, E1   +43.653, E3 +74975.207}
SPL {X  -154.385, Y  +346.786, Z    +0.000, E1   +43.356, E3 +74993.619}
SPL {X  -152.146, Y  +339.286, Z    +0.000, E1   +42.904, E3 +75012.254}
SPL {X  -149.854, Y  +332.731, Z    +0.000, E1   +42.474, E3 +75028.781}
SPL {X  -145.635, Y  +322.541, Z    +0.000, E1   +36.397, E3 +75104.740}
ENDSPLINE

SPLINE
SPL {X  -156.682, Y  +356.385, Z    +0.000, E1   +19.033, E3 +75163.047}
SPL {X  -159.526, Y  +376.492, Z    +0.000, E1    +8.067, E3 +75172.956}
SPL {X  -159.961, Y  +385.275, Z    +0.000, E1    +2.550, E3 +75174.994}
SPL {X  -160.000, Y  +390.345, Z    +0.000, E1    -1.188, E3 +75175.720}
SPL {X  -160.000, Y  +395.838, Z    +0.000, E1    -6.211, E3 +75176.664}
SPL {X  -160.000, Y  +403.277, Z    +0.000, E1   -14.057, E3 +75178.615}
SPL {X  -160.000, Y  +414.316, Z    +0.000, E1   -24.810, E3 +75183.688}
SPL {X  -160.000, Y  +442.604, Z    +0.000, E1   -40.161, E3 +75205.822}
SPL {X  -160.000, Y  +482.867, Z    +0.000, E1   -45.148, E3 +75266.038}
SPL {X  -160.000, Y  +494.769, Z    +0.000, E1   -45.151, E3 +75291.257}
SPL {X  -160.000, Y  +505.761, Z    +0.000, E1   -45.118, E3 +75314.571}
SPL {X  -160.000, Y  +517.347, Z    +0.000, E1   -45.173, E3 +75339.009}
SPL {X  -160.000, Y  +529.298, Z    +0.000, E1   -45.138, E3 +75364.392}
SPL {X  -160.000, Y  +540.664, Z    +0.000, E1   -45.139, E3 +75388.470}
SPL {X  -160.000, Y  +552.011, Z    +0.000, E1   -45.139, E3 +75412.506}
SPL {X  -160.000, Y  +563.667, Z    +0.000, E1   -45.146, E3 +75437.186}
SPL {X  -160.000, Y  +574.965, Z    +0.000, E1   -45.125, E3 +75461.162}
SPL {X  -160.000, Y  +585.644, Z    +0.000, E1   -45.117, E3 +75483.802}
SPL {X  -160.000, Y  +596.819, Z    +0.000, E1   -45.144, E3 +75507.444}
SPL {X  -160.000, Y  +608.165, Z    +0.000, E1   -45.120, E3 +75531.518}
SPL {X  -160.000, Y  +619.270, Z    +0.000, E1   -45.132, E3 +75555.021}
SPL {X  -160.000, Y  +629.968, Z    +0.000, E1   -45.117, E3 +75577.687}
SPL {X  -160.000, Y  +640.750, Z    +0.000, E1   -45.131, E3 +75600.510}
SPL {X  -160.000, Y  +651.429, Z    +0.000, E1   -45.117, E3 +75623.151}
SPL {X  -160.000, Y  +662.434, Z    +0.000, E1   -45.129, E3 +75646.495}
SPL {X  -159.992, Y  +673.110, Z    +0.000, E1   -45.097, E3 +75669.188}
SPL {X  -159.521, Y  +683.874, Z    +0.000, E1   -45.054, E3 +75692.443}
SPL {X  -158.435, Y  +693.823, Z    +0.000, E1   -44.810, E3 +75714.747}
SPL {X  -156.807, Y  +703.304, Z    +0.000, E1   -44.558, E3 +75736.468}
SPL {X  -154.802, Y  +711.950, Z    +0.000, E1   -44.141, E3 +75756.928}
SPL {X  -152.641, Y  +719.464, Z    +0.000, E1   -43.749, E3 +75775.044}
SPL {X  -149.826, Y  +727.645, Z    +0.000, E1   -43.252, E3 +75795.146}
SPL {X  -145.307, Y  +738.478, Z    +0.000, E1   -36.676, E3 +75875.214}
ENDSPLINE

SPLINE
SPL {X  -155.601, Y  +708.762, Z    +0.000, E1   -21.463, E3 +75930.001}
SPL {X  -158.549, Y  +693.002, Z    +0.000, E1   -13.406, E3 +75938.991}
SPL {X  -159.716, Y  +681.031, Z    +0.000, E1    -6.529, E3 +75943.142}
SPL {X  -160.000, Y  +671.641, Z    +0.000, E1    -0.547, E3 +75944.858}
SPL {X  -160.000, Y  +665.424, Z    +0.000, E1    +5.044, E3 +75945.806}
SPL {X  -160.000, Y  +658.015, Z    +0.000, E1   +12.630, E3 +75947.724}
SPL {X  -160.000, Y  +645.110, Z    +0.000, E1   +25.142, E3 +75953.524}
SPL {X  -160.000, Y  +611.664, Z    +0.000, E1   +41.262, E3 +75983.254}
SPL {X  -160.000, Y  +581.433, Z    +0.000, E1   +44.103, E3 +76032.990}
SPL {X  -160.000, Y  +572.090, Z    +0.000, E1   +44.120, E3 +76053.455}
SPL {X  -160.000, Y  +563.431, Z    +0.000, E1   +44.084, E3 +76072.508}
SPL {X  -160.000, Y  +556.107, Z    +0.000, E1   +44.076, E3 +76088.576}
SPL {X  -160.000, Y  +549.181, Z    +0.000, E1   +44.079, E3 +76103.736}
SPL {X  -160.000, Y  +542.413, Z    +0.000, E1   +44.088, E3 +76118.570}
SPL {X  -160.000, Y  +534.609, Z    +0.000, E1   +44.095, E3 +76135.680}
SPL {X  -160.000, Y  +527.457, Z    +0.000, E1   +44.070, E3 +76151.390}
SPL {X  -160.000, Y  +520.912, Z    +0.000, E1   +44.079, E3 +76165.731}
SPL {X  -160.000, Y  +514.086, Z    +0.000, E1   +44.081, E3 +76180.680}
SPL {X  -160.000, Y  +507.208, Z    +0.000, E1   +44.082, E3 +76195.756}
SPL {X  -160.000, Y  +499.184, Z    +0.000, E1   +44.113, E3 +76213.314}
ENDSPLINE

SPLINE
SPL {X  -160.000, Y  +503.824, Z    +0.000, E1   +39.488, E3 +76229.363}
ENDSPLINE

SPLINE
SPL {X  -160.000, Y  +499.279, Z    +0.000, E1   +38.981, E3 +76244.353}
SPL {X  -160.000, Y  +490.068, Z    +0.000, E1   +40.198, E3 +76260.657}
SPL {X  -160.000, Y  +481.368, Z    +0.000, E1   +41.274, E3 +76275.647}
SPL {X  -160.000, Y  +470.910, Z    +0.000, E1   +42.658, E3 +76292.155}
SPL {X  -160.000, Y  +460.219, Z    +0.000, E1   +43.912, E3 +76308.776}
SPL {X  -160.000, Y  +451.951, Z    +0.000, E1   +44.355, E3 +76324.341}
SPL {X  -160.000, Y  +442.331, Z    +0.000, E1   +44.390, E3 +76345.206}
SPL {X  -160.000, Y  +433.037, Z    +0.000, E1   +44.348, E3 +76365.480}
SPL {X  -160.000, Y  +424.435, Z    +0.000, E1   +44.358, E3 +76384.148}
SPL {X  -160.000, Y  +416.015, Z    +0.000, E1   +44.348, E3 +76402.468}
SPL {X  -160.000, Y  +407.167, Z    +0.000, E1   +44.365, E3 +76421.679}
SPL {X  -160.000, Y  +397.599, Z    +0.000, E1   +44.371, E3 +76442.487}
SPL {X  -160.000, Y  +388.533, Z    +0.000, E1   +44.340, E3 +76462.262}
SPL {X  -159.759, Y  +380.021, Z    +0.000, E1   +44.311, E3 +76480.994}
SPL {X  -159.014, Y  +371.065, Z    +0.000, E1   +44.193, E3 +76501.232}
SPL {X  -157.745, Y  +362.030, Z    +0.000, E1   +43.965, E3 +76522.214}
SPL {X  -156.258, Y  +354.400, Z    +0.000, E1   +43.653, E3 +76540.422}
SPL {X  -154.385, Y  +346.786, Z    +0.000, E1   +43.356, E3 +76558.833}
SPL {X  -152.146, Y  +339.286, Z    +0.000, E1   +42.904, E3 +76577.468}
SPL {X  -149.854, Y  +332.731, Z    +0.000, E1   +42.474, E3 +76593.996}
SPL {X  -145.635, Y  +322.541, Z    +0.000, E1   +36.397, E3 +76669.955}
ENDSPLINE

SPLINE
SPL {X  -156.682, Y  +356.385, Z    +0.000, E1   +19.033, E3 +76728.261}
SPL {X  -159.526, Y  +376.492, Z    +0.000, E1    +8.067, E3 +76738.170}
SPL {X  -159.961, Y  +385.275, Z    +0.000, E1    +2.550, E3 +76740.208}
SPL {X  -160.000, Y  +390.345, Z    +0.000, E1    -1.188, E3 +76740.934}
SPL {X  -160.000, Y  +395.838, Z    +0.000, E1    -6.211, E3 +76741.878}
SPL {X  -160.000, Y  +403.277, Z    +0.000, E1   -14.057, E3 +76743.829}
SPL {X  -160.000, Y  +414.316, Z    +0.000, E1   -24.810, E3 +76748.902}
SPL {X  -160.000, Y  +442.604, Z    +0.000, E1   -40.161, E3 +76771.036}
SPL {X  -160.000, Y  +482.867, Z    +0.000, E1   -45.148, E3 +76831.252}
SPL {X  -160.000, Y  +494.769, Z    +0.000, E1   -45.151, E3 +76856.471}
SPL {X  -160.000, Y  +505.761, Z    +0.000, E1   -45.118, E3 +76879.785}
SPL {X  -160.000, Y  +517.347, Z    +0.000, E1   -45.173, E3 +76904.223}
SPL {X  -160.000, Y  +529.298, Z    +0.000, E1   -45.138, E3 +76929.606}
SPL {X  -160.000, Y  +540.664, Z    +0.000, E1   -45.139, E3 +76953.684}
SPL {X  -160.000, Y  +552.011, Z    +0.000, E1   -45.139, E3 +76977.720}
SPL {X  -160.000, Y  +563.667, Z    +0.000, E1   -45.146, E3 +77002.401}
SPL {X  -160.000, Y  +574.965, Z    +0.000, E1   -45.125, E3 +77026.376}
SPL {X  -160.000, Y  +585.644, Z    +0.000, E1   -45.117, E3 +77049.016}
SPL {X  -160.000, Y  +596.819, Z    +0.000, E1   -45.144, E3 +77072.658}
SPL {X  -160.000, Y  +608.165, Z    +0.000, E1   -45.120, E3 +77096.732}
SPL {X  -160.000, Y  +619.270, Z    +0.000, E1   -45.132, E3 +77120.235}
SPL {X  -160.000, Y  +629.968, Z    +0.000, E1   -45.117, E3 +77142.901}
SPL {X  -160.000, Y  +640.750, Z    +0.000, E1   -45.131, E3 +77165.724}
SPL {X  -160.000, Y  +651.429, Z    +0.000, E1   -45.117, E3 +77188.365}
SPL {X  -160.000, Y  +662.434, Z    +0.000, E1   -45.129, E3 +77211.709}
SPL {X  -159.992, Y  +673.110, Z    +0.000, E1   -45.097, E3 +77234.402}
SPL {X  -159.521, Y  +683.874, Z    +0.000, E1   -45.054, E3 +77257.657}
SPL {X  -158.435, Y  +693.823, Z    +0.000, E1   -44.810, E3 +77279.961}
SPL {X  -156.807, Y  +703.304, Z    +0.000, E1   -44.558, E3 +77301.682}
SPL {X  -154.802, Y  +711.950, Z    +0.000, E1   -44.141, E3 +77322.142}
SPL {X  -152.641, Y  +719.464, Z    +0.000, E1   -43.749, E3 +77340.258}
SPL {X  -149.826, Y  +727.645, Z    +0.000, E1   -43.252, E3 +77360.361}
SPL {X  -145.307, Y  +738.478, Z    +0.000, E1   -36.676, E3 +77440.428}
ENDSPLINE

SPLINE
SPL {X  -155.601, Y  +708.762, Z    +0.000, E1   -21.463, E3 +77495.215}
SPL {X  -158.549, Y  +693.002, Z    +0.000, E1   -13.406, E3 +77504.206}
SPL {X  -159.716, Y  +681.031, Z    +0.000, E1    -6.529, E3 +77508.356}
SPL {X  -160.000, Y  +671.641, Z    +0.000, E1    -0.547, E3 +77510.072}
SPL {X  -160.000, Y  +665.424, Z    +0.000, E1    +5.044, E3 +77511.021}
SPL {X  -160.000, Y  +658.015, Z    +0.000, E1   +12.630, E3 +77512.938}
SPL {X  -160.000, Y  +645.110, Z    +0.000, E1   +25.142, E3 +77518.738}
SPL {X  -160.000, Y  +611.664, Z    +0.000, E1   +41.262, E3 +77548.468}
SPL {X  -160.000, Y  +581.433, Z    +0.000, E1   +44.103, E3 +77598.205}
SPL {X  -160.000, Y  +572.090, Z    +0.000, E1   +44.120, E3 +77618.669}
SPL {X  -160.000, Y  +563.431, Z    +0.000, E1   +44.084, E3 +77637.722}
SPL {X  -160.000, Y  +556.107, Z    +0.000, E1   +44.076, E3 +77653.791}
SPL {X  -160.000, Y  +549.181, Z    +0.000, E1   +44.079, E3 +77668.950}
SPL {X  -160.000, Y  +542.413, Z    +0.000, E1   +44.088, E3 +77683.784}
SPL {X  -160.000, Y  +534.609, Z    +0.000, E1   +44.095, E3 +77700.894}
SPL {X  -160.000, Y  +527.457, Z    +0.000, E1   +44.070, E3 +77716.605}
SPL {X  -160.000, Y  +520.912, Z    +0.000, E1   +44.079, E3 +77730.945}
SPL {X  -160.000, Y  +514.086, Z    +0.000, E1   +44.081, E3 +77745.894}
SPL {X  -160.000, Y  +507.208, Z    +0.000, E1   +44.082, E3 +77760.970}
SPL {X  -160.000, Y  +499.184, Z    +0.000, E1   +44.113, E3 +77778.528}
ENDSPLINE

SPLINE
SPL {X  -160.000, Y  +503.824, Z    +0.000, E1   +39.488, E3 +77794.577}
ENDSPLINE

SPLINE
SPL {X  -160.000, Y  +499.279, Z    +0.000, E1   +38.981, E3 +77809.567}
SPL {X  -160.000, Y  +490.068, Z    +0.000, E1   +40.198, E3 +77825.871}
SPL {X  -160.000, Y  +481.368, Z    +0.000, E1   +41.274, E3 +77840.861}
SPL {X  -160.000, Y  +470.910, Z    +0.000, E1   +42.658, E3 +77857.370}
SPL {X  -160.000, Y  +460.219, Z    +0.000, E1   +43.912, E3 +77873.990}
SPL {X  -160.000, Y  +451.951, Z    +0.000, E1   +44.355, E3 +77889.556}
SPL {X  -160.000, Y  +442.331, Z    +0.000, E1   +44.390, E3 +77910.420}
SPL {X  -160.000, Y  +433.037, Z    +0.000, E1   +44.348, E3 +77930.694}
SPL {X  -160.000, Y  +424.435, Z    +0.000, E1   +44.358, E3 +77949.362}
SPL {X  -160.000, Y  +416.015, Z    +0.000, E1   +44.348, E3 +77967.682}
SPL {X  -160.000, Y  +407.167, Z    +0.000, E1   +44.365, E3 +77986.893}
SPL {X  -160.000, Y  +397.599, Z    +0.000, E1   +44.371, E3 +78007.701}
SPL {X  -160.000, Y  +388.533, Z    +0.000, E1   +44.340, E3 +78027.476}
SPL {X  -159.759, Y  +380.021, Z    +0.000, E1   +44.311, E3 +78046.208}
SPL {X  -159.014, Y  +371.065, Z    +0.000, E1   +44.193, E3 +78066.446}
SPL {X  -157.745, Y  +362.030, Z    +0.000, E1   +43.965, E3 +78087.428}
SPL {X  -156.258, Y  +354.400, Z    +0.000, E1   +43.653, E3 +78105.636}
SPL {X  -154.385, Y  +346.786, Z    +0.000, E1   +43.356, E3 +78124.047}
SPL {X  -152.146, Y  +339.286, Z    +0.000, E1   +42.904, E3 +78142.682}
SPL {X  -149.854, Y  +332.731, Z    +0.000, E1   +42.474, E3 +78159.210}
SPL {X  -145.635, Y  +322.541, Z    +0.000, E1   +36.397, E3 +78235.169}
ENDSPLINE

SPLINE
SPL {X  -156.682, Y  +356.385, Z    +0.000, E1   +19.033, E3 +78293.475}
SPL {X  -159.526, Y  +376.492, Z    +0.000, E1    +8.067, E3 +78303.384}
SPL {X  -159.961, Y  +385.275, Z    +0.000, E1    +2.550, E3 +78305.422}
SPL {X  -160.000, Y  +390.345, Z    +0.000, E1    -1.188, E3 +78306.148}
SPL {X  -160.000, Y  +395.838, Z    +0.000, E1    -6.211, E3 +78307.092}
SPL {X  -160.000, Y  +403.277, Z    +0.000, E1   -14.057, E3 +78309.043}
SPL {X  -160.000, Y  +414.316, Z    +0.000, E1   -24.810, E3 +78314.116}
SPL {X  -160.000, Y  +442.604, Z    +0.000, E1   -40.161, E3 +78336.250}
SPL {X  -160.000, Y  +482.867, Z    +0.000, E1   -45.148, E3 +78396.466}
SPL {X  -160.000, Y  +494.769, Z    +0.000, E1   -45.151, E3 +78421.686}
SPL {X  -160.000, Y  +505.761, Z    +0.000, E1   -45.118, E3 +78445.000}
SPL {X  -160.000, Y  +517.347, Z    +0.000, E1   -45.173, E3 +78469.437}
SPL {X  -160.000, Y  +529.298, Z    +0.000, E1   -45.138, E3 +78494.821}
SPL {X  -160.000, Y  +540.664, Z    +0.000, E1   -45.139, E3 +78518.898}
SPL {X  -160.000, Y  +552.011, Z    +0.000, E1   -45.139, E3 +78542.934}
SPL {X  -160.000, Y  +563.667, Z    +0.000, E1   -45.146, E3 +78567.615}
SPL {X  -160.000, Y  +574.965, Z    +0.000, E1   -45.125, E3 +78591.590}
SPL {X  -160.000, Y  +585.644, Z    +0.000, E1   -45.117, E3 +78614.230}
SPL {X  -160.000, Y  +596.819, Z    +0.000, E1   -45.144, E3 +78637.872}
SPL {X  -160.000, Y  +608.165, Z    +0.000, E1   -45.120, E3 +78661.946}
SPL {X  -160.000, Y  +619.270, Z    +0.000, E1   -45.132, E3 +78685.449}
SPL {X  -160.000, Y  +629.968, Z    +0.000, E1   -45.117, E3 +78708.115}
SPL {X  -160.000, Y  +640.750, Z    +0.000, E1   -45.131, E3 +78730.938}
SPL {X  -160.000, Y  +651.429, Z    +0.000, E1   -45.117, E3 +78753.579}
SPL {X  -160.000, Y  +662.434, Z    +0.000, E1   -45.129, E3 +78776.923}
SPL {X  -159.992, Y  +673.110, Z    +0.000, E1   -45.097, E3 +78799.616}
SPL {X  -159.521, Y  +683.874, Z    +0.000, E1   -45.054, E3 +78822.871}
SPL {X  -158.435, Y  +693.823, Z    +0.000, E1   -44.810, E3 +78845.175}
SPL {X  -156.807, Y  +703.304, Z    +0.000, E1   -44.558, E3 +78866.896}
SPL {X  -154.802, Y  +711.950, Z    +0.000, E1   -44.141, E3 +78887.356}
SPL {X  -152.641, Y  +719.464, Z    +0.000, E1   -43.749, E3 +78905.472}
SPL {X  -149.826, Y  +727.645, Z    +0.000, E1   -43.252, E3 +78925.575}
SPL {X  -145.307, Y  +738.478, Z    +0.000, E1   -36.676, E3 +79005.642}
ENDSPLINE

SPLINE
SPL {X  -155.601, Y  +708.762, Z    +0.000, E1   -21.463, E3 +79060.429}
SPL {X  -158.549, Y  +693.002, Z    +0.000, E1   -13.406, E3 +79069.420}
SPL {X  -159.716, Y  +681.031, Z    +0.000, E1    -6.529, E3 +79073.570}
SPL {X  -160.000, Y  +671.641, Z    +0.000, E1    -0.547, E3 +79075.287}
SPL {X  -160.000, Y  +665.424, Z    +0.000, E1    +5.044, E3 +79076.235}
SPL {X  -160.000, Y  +658.015, Z    +0.000, E1   +12.630, E3 +79078.153}
SPL {X  -160.000, Y  +645.110, Z    +0.000, E1   +25.142, E3 +79083.953}
SPL {X  -160.000, Y  +611.664, Z    +0.000, E1   +41.262, E3 +79113.682}
SPL {X  -160.000, Y  +581.433, Z    +0.000, E1   +44.103, E3 +79163.419}
SPL {X  -160.000, Y  +572.090, Z    +0.000, E1   +44.120, E3 +79183.883}
SPL {X  -160.000, Y  +563.431, Z    +0.000, E1   +44.084, E3 +79202.936}
SPL {X  -160.000, Y  +556.107, Z    +0.000, E1   +44.076, E3 +79219.005}
SPL {X  -160.000, Y  +549.181, Z    +0.000, E1   +44.079, E3 +79234.164}
SPL {X  -160.000, Y  +542.413, Z    +0.000, E1   +44.088, E3 +79248.998}
SPL {X  -160.000, Y  +534.609, Z    +0.000, E1   +44.095, E3 +79266.108}
SPL {X  -160.000, Y  +527.457, Z    +0.000, E1   +44.070, E3 +79281.819}
SPL {X  -160.000, Y  +520.912, Z    +0.000, E1   +44.079, E3 +79296.160}
SPL {X  -160.000, Y  +514.086, Z    +0.000, E1   +44.081, E3 +79311.108}
SPL {X  -160.000, Y  +507.208, Z    +0.000, E1   +44.082, E3 +79326.184}
SPL {X  -160.000, Y  +499.184, Z    +0.000, E1   +44.113, E3 +79343.742}
ENDSPLINE

SPLINE
SPL {X  -160.000, Y  +503.824, Z    +0.000, E1   +39.488, E3 +79359.791}
ENDSPLINE

SPLINE
SPL {X  -160.000, Y  +499.279, Z    +0.000, E1   +38.981, E3 +79374.781}
SPL {X  -160.000, Y  +490.068, Z    +0.000, E1   +40.198, E3 +79391.085}
SPL {X  -160.000, Y  +481.368, Z    +0.000, E1   +41.274, E3 +79406.075}
SPL {X  -160.000, Y  +470.910, Z    +0.000, E1   +42.658, E3 +79422.584}
SPL {X  -160.000, Y  +460.219, Z    +0.000, E1   +43.912, E3 +79439.204}
SPL {X  -160.000, Y  +451.951, Z    +0.000, E1   +44.355, E3 +79454.770}
SPL {X  -160.000, Y  +442.331, Z    +0.000, E1   +44.390, E3 +79475.634}
SPL {X  -160.000, Y  +433.037, Z    +0.000, E1   +44.348, E3 +79495.908}
SPL {X  -160.000, Y  +424.435, Z    +0.000, E1   +44.358, E3 +79514.576}
SPL {X  -160.000, Y  +416.015, Z    +0.000, E1   +44.348, E3 +79532.896}
SPL {X  -160.000, Y  +407.167, Z    +0.000, E1   +44.365, E3 +79552.107}
SPL {X  -160.000, Y  +397.599, Z    +0.000, E1   +44.371, E3 +79572.915}
SPL {X  -160.000, Y  +388.533, Z    +0.000, E1   +44.340, E3 +79592.690}
SPL {X  -159.759, Y  +380.021, Z    +0.000, E1   +44.311, E3 +79611.422}
SPL {X  -159.014, Y  +371.065, Z    +0.000, E1   +44.193, E3 +79631.660}
SPL {X  -157.745, Y  +362.030, Z    +0.000, E1   +43.965, E3 +79652.642}
SPL {X  -156.258, Y  +354.400, Z    +0.000, E1   +43.653, E3 +79670.850}
SPL {X  -154.385, Y  +346.786, Z    +0.000, E1   +43.356, E3 +79689.262}
SPL {X  -152.146, Y  +339.286, Z    +0.000, E1   +42.904, E3 +79707.896}
SPL {X  -149.854, Y  +332.731, Z    +0.000, E1   +42.474, E3 +79724.424}
SPL {X  -145.635, Y  +322.541, Z    +0.000, E1   +36.397, E3 +79800.383}
ENDSPLINE

SPLINE
SPL {X  -156.682, Y  +356.385, Z    +0.000, E1   +19.033, E3 +79858.689}
SPL {X  -159.526, Y  +376.492, Z    +0.000, E1    +8.067, E3 +79868.598}
SPL {X  -159.961, Y  +385.275, Z    +0.000, E1    +2.550, E3 +79870.637}
SPL {X  -160.000, Y  +390.345, Z    +0.000, E1    -1.188, E3 +79871.363}
SPL {X  -160.000, Y  +395.838, Z    +0.000, E1    -6.211, E3 +79872.306}
SPL {X  -160.000, Y  +403.277, Z    +0.000, E1   -14.057, E3 +79874.257}
SPL {X  -160.000, Y  +414.316, Z    +0.000, E1   -24.810, E3 +79879.330}
SPL {X  -160.000, Y  +442.604, Z    +0.000, E1   -40.161, E3 +79901.464}
SPL {X  -160.000, Y  +482.867, Z    +0.000, E1   -45.148, E3 +79961.680}
SPL {X  -160.000, Y  +494.769, Z    +0.000, E1   -45.151, E3 +79986.900}
SPL {X  -160.000, Y  +505.761, Z    +0.000, E1   -45.118, E3 +80010.214}
SPL {X  -160.000, Y  +517.347, Z    +0.000, E1   -45.173, E3 +80034.651}
SPL {X  -160.000, Y  +529.298, Z    +0.000, E1   -45.138, E3 +80060.035}
SPL {X  -160.000, Y  +540.664, Z    +0.000, E1   -45.139, E3 +80084.113}
SPL {X  -160.000, Y  +552.011, Z    +0.000, E1   -45.139, E3 +80108.148}
SPL {X  -160.000, Y  +563.667, Z    +0.000, E1   -45.146, E3 +80132.829}
SPL {X  -160.000, Y  +574.965, Z    +0.000, E1   -45.125, E3 +80156.804}
SPL {X  -160.000, Y  +585.644, Z    +0.000, E1   -45.117, E3 +80179.444}
SPL {X  -160.000, Y  +596.819, Z    +0.000, E1   -45.144, E3 +80203.086}
SPL {X  -160.000, Y  +608.165, Z    +0.000, E1   -45.120, E3 +80227.160}
SPL {X  -160.000, Y  +619.270, Z    +0.000, E1   -45.132, E3 +80250.663}
SPL {X  -160.000, Y  +629.968, Z    +0.000, E1   -45.117, E3 +80273.329}
SPL {X  -160.000, Y  +640.750, Z    +0.000, E1   -45.131, E3 +80296.152}
SPL {X  -160.000, Y  +651.429, Z    +0.000, E1   -45.117, E3 +80318.794}
SPL {X  -160.000, Y  +662.434, Z    +0.000, E1   -45.129, E3 +80342.137}
SPL {X  -159.992, Y  +673.110, Z    +0.000, E1   -45.097, E3 +80364.830}
SPL {X  -159.521, Y  +683.874, Z    +0.000, E1   -45.054, E3 +80388.085}
SPL {X  -158.435, Y  +693.823, Z    +0.000, E1   -44.810, E3 +80410.390}
SPL {X  -156.807, Y  +703.304, Z    +0.000, E1   -44.558, E3 +80432.110}
SPL {X  -154.802, Y  +711.950, Z    +0.000, E1   -44.141, E3 +80452.570}
SPL {X  -152.641, Y  +719.464, Z    +0.000, E1   -43.749, E3 +80470.686}
SPL {X  -149.826, Y  +727.645, Z    +0.000, E1   -43.252, E3 +80490.789}
SPL {X  -145.307, Y  +738.478, Z    +0.000, E1   -36.676, E3 +80570.856}
ENDSPLINE

SPLINE
SPL {X  -155.601, Y  +708.762, Z    +0.000, E1   -21.463, E3 +80625.643}
SPL {X  -158.549, Y  +693.002, Z    +0.000, E1   -13.406, E3 +80634.634}
SPL {X  -159.716, Y  +681.031, Z    +0.000, E1    -6.529, E3 +80638.784}
SPL {X  -160.000, Y  +671.641, Z    +0.000, E1    -0.547, E3 +80640.501}
SPL {X  -160.000, Y  +665.424, Z    +0.000, E1    +5.044, E3 +80641.449}
SPL {X  -160.000, Y  +658.015, Z    +0.000, E1   +12.630, E3 +80643.367}
SPL {X  -160.000, Y  +645.110, Z    +0.000, E1   +25.142, E3 +80649.167}
SPL {X  -160.000, Y  +611.664, Z    +0.000, E1   +41.262, E3 +80678.896}
SPL {X  -160.000, Y  +581.433, Z    +0.000, E1   +44.103, E3 +80728.633}
SPL {X  -160.000, Y  +572.090, Z    +0.000, E1   +44.120, E3 +80749.097}
SPL {X  -160.000, Y  +563.431, Z    +0.000, E1   +44.084, E3 +80768.151}
SPL {X  -160.000, Y  +556.107, Z    +0.000, E1   +44.076, E3 +80784.219}
SPL {X  -160.000, Y  +549.181, Z    +0.000, E1   +44.079, E3 +80799.378}
SPL {X  -160.000, Y  +542.413, Z    +0.000, E1   +44.088, E3 +80814.212}
SPL {X  -160.000, Y  +534.609, Z    +0.000, E1   +44.095, E3 +80831.322}
SPL {X  -160.000, Y  +527.457, Z    +0.000, E1   +44.070, E3 +80847.033}
SPL {X  -160.000, Y  +520.912, Z    +0.000, E1   +44.079, E3 +80861.374}
SPL {X  -160.000, Y  +514.086, Z    +0.000, E1   +44.081, E3 +80876.322}
SPL {X  -160.000, Y  +507.208, Z    +0.000, E1   +44.082, E3 +80891.398}
SPL {X  -160.000, Y  +499.184, Z    +0.000, E1   +44.113, E3 +80908.957}
ENDSPLINE

SPLINE
SPL {X  -160.000, Y  +503.824, Z    +0.000, E1   +39.488, E3 +80925.005}
ENDSPLINE

SPLINE
SPL {X  -160.000, Y  +499.279, Z    +0.000, E1   +38.981, E3 +80939.995}
SPL {X  -160.000, Y  +490.068, Z    +0.000, E1   +40.198, E3 +80956.299}
SPL {X  -160.000, Y  +481.368, Z    +0.000, E1   +41.274, E3 +80971.289}
SPL {X  -160.000, Y  +470.910, Z    +0.000, E1   +42.658, E3 +80987.798}
SPL {X  -160.000, Y  +460.219, Z    +0.000, E1   +43.912, E3 +81004.418}
SPL {X  -160.000, Y  +451.951, Z    +0.000, E1   +44.355, E3 +81019.984}
SPL {X  -160.000, Y  +442.331, Z    +0.000, E1   +44.390, E3 +81040.848}
SPL {X  -160.000, Y  +433.037, Z    +0.000, E1   +44.348, E3 +81061.122}
SPL {X  -160.000, Y  +424.435, Z    +0.000, E1   +44.358, E3 +81079.791}
SPL {X  -160.000, Y  +416.015, Z    +0.000, E1   +44.348, E3 +81098.111}
SPL {X  -160.000, Y  +407.167, Z    +0.000, E1   +44.365, E3 +81117.321}
SPL {X  -160.000, Y  +397.599, Z    +0.000, E1   +44.371, E3 +81138.130}
SPL {X  -160.000, Y  +388.533, Z    +0.000, E1   +44.340, E3 +81157.904}
SPL {X  -159.759, Y  +380.021, Z    +0.000, E1   +44.311, E3 +81176.637}
SPL {X  -159.014, Y  +371.065, Z    +0.000, E1   +44.193, E3 +81196.875}
SPL {X  -157.745, Y  +362.030, Z    +0.000, E1   +43.965, E3 +81217.857}
SPL {X  -156.258, Y  +354.400, Z    +0.000, E1   +43.653, E3 +81236.064}
SPL {X  -154.385, Y  +346.786, Z    +0.000, E1   +43.356, E3 +81254.476}
SPL {X  -152.146, Y  +339.286, Z    +0.000, E1   +42.904, E3 +81273.110}
SPL {X  -149.854, Y  +332.731, Z    +0.000, E1   +42.474, E3 +81289.638}
SPL {X  -145.635, Y  +322.541, Z    +0.000, E1   +36.397, E3 +81365.597}
ENDSPLINE

SPLINE
SPL {X  -156.682, Y  +356.385, Z    +0.000, E1   +19.033, E3 +81423.903}
SPL {X  -159.526, Y  +376.492, Z    +0.000, E1    +8.067, E3 +81433.812}
SPL {X  -159.961, Y  +385.275, Z    +0.000, E1    +2.550, E3 +81435.851}
SPL {X  -160.000, Y  +390.345, Z    +0.000, E1    -1.188, E3 +81436.577}
SPL {X  -160.000, Y  +395.838, Z    +0.000, E1    -6.211, E3 +81437.520}
SPL {X  -160.000, Y  +403.277, Z    +0.000, E1   -14.057, E3 +81439.471}
SPL {X  -160.000, Y  +414.316, Z    +0.000, E1   -24.810, E3 +81444.544}
SPL {X  -160.000, Y  +442.604, Z    +0.000, E1   -40.161, E3 +81466.678}
SPL {X  -160.000, Y  +482.867, Z    +0.000, E1   -45.148, E3 +81526.895}
SPL {X  -160.000, Y  +494.769, Z    +0.000, E1   -45.151, E3 +81552.114}
SPL {X  -160.000, Y  +505.761, Z    +0.000, E1   -45.118, E3 +81575.428}
SPL {X  -160.000, Y  +517.347, Z    +0.000, E1   -45.173, E3 +81599.865}
SPL {X  -160.000, Y  +529.298, Z    +0.000, E1   -45.138, E3 +81625.249}
SPL {X  -160.000, Y  +540.664, Z    +0.000, E1   -45.139, E3 +81649.327}
SPL {X  -160.000, Y  +552.011, Z    +0.000, E1   -45.139, E3 +81673.363}
SPL {X  -160.000, Y  +563.667, Z    +0.000, E1   -45.146, E3 +81698.043}
SPL {X  -160.000, Y  +574.965, Z    +0.000, E1   -45.125, E3 +81722.019}
SPL {X  -160.000, Y  +585.644, Z    +0.000, E1   -45.117, E3 +81744.659}
SPL {X  -160.000, Y  +596.819, Z    +0.000, E1   -45.144, E3 +81768.300}
SPL {X  -160.000, Y  +608.165, Z    +0.000, E1   -45.120, E3 +81792.375}
SPL {X  -160.000, Y  +619.270, Z    +0.000, E1   -45.132, E3 +81815.877}
SPL {X  -160.000, Y  +629.968, Z    +0.000, E1   -45.117, E3 +81838.543}
SPL {X  -160.000, Y  +640.750, Z    +0.000, E1   -45.131, E3 +81861.366}
SPL {X  -160.000, Y  +651.429, Z    +0.000, E1   -45.117, E3 +81884.008}
SPL {X  -160.000, Y  +662.434, Z    +0.000, E1   -45.129, E3 +81907.352}
SPL {X  -159.992, Y  +673.110, Z    +0.000, E1   -45.097, E3 +81930.044}
SPL {X  -159.521, Y  +683.874, Z    +0.000, E1   -45.054, E3 +81953.299}
SPL {X  -158.435, Y  +693.823, Z    +0.000, E1   -44.810, E3 +81975.604}
SPL {X  -156.807, Y  +703.304, Z    +0.000, E1   -44.558, E3 +81997.324}
SPL {X  -154.802, Y  +711.950, Z    +0.000, E1   -44.141, E3 +82017.784}
SPL {X  -152.641, Y  +719.464, Z    +0.000, E1   -43.749, E3 +82035.900}
SPL {X  -149.826, Y  +727.645, Z    +0.000, E1   -43.252, E3 +82056.003}
SPL {X  -145.307, Y  +738.478, Z    +0.000, E1   -36.676, E3 +82136.071}
ENDSPLINE

SPLINE
SPL {X  -155.601, Y  +708.762, Z    +0.000, E1   -21.463, E3 +82190.857}
SPL {X  -158.549, Y  +693.002, Z    +0.000, E1   -13.406, E3 +82199.848}
SPL {X  -159.716, Y  +681.031, Z    +0.000, E1    -6.529, E3 +82203.998}
SPL {X  -160.000, Y  +671.641, Z    +0.000, E1    -0.547, E3 +82205.715}
SPL {X  -160.000, Y  +665.424, Z    +0.000, E1    +5.044, E3 +82206.663}
SPL {X  -160.000, Y  +658.015, Z    +0.000, E1   +12.630, E3 +82208.581}
SPL {X  -160.000, Y  +645.110, Z    +0.000, E1   +25.142, E3 +82214.381}
SPL {X  -160.000, Y  +611.664, Z    +0.000, E1   +41.262, E3 +82244.110}
SPL {X  -160.000, Y  +581.433, Z    +0.000, E1   +44.103, E3 +82293.847}
SPL {X  -160.000, Y  +572.090, Z    +0.000, E1   +44.120, E3 +82314.311}
SPL {X  -160.000, Y  +563.431, Z    +0.000, E1   +44.084, E3 +82333.365}
SPL {X  -160.000, Y  +556.107, Z    +0.000, E1   +44.076, E3 +82349.433}
SPL {X  -160.000, Y  +549.181, Z    +0.000, E1   +44.079, E3 +82364.593}
SPL {X  -160.000, Y  +542.413, Z    +0.000, E1   +44.088, E3 +82379.427}
SPL {X  -160.000, Y  +534.609, Z    +0.000, E1   +44.095, E3 +82396.537}
SPL {X  -160.000, Y  +527.457, Z    +0.000, E1   +44.070, E3 +82412.247}
SPL {X  -160.000, Y  +520.912, Z    +0.000, E1   +44.079, E3 +82426.588}
SPL {X  -160.000, Y  +514.086, Z    +0.000, E1   +44.081, E3 +82441.536}
SPL {X  -160.000, Y  +507.208, Z    +0.000, E1   +44.082, E3 +82456.613}
SPL {X  -160.000, Y  +499.184, Z    +0.000, E1   +44.113, E3 +82474.171}
ENDSPLINE

SPLINE
SPL {X  -160.000, Y  +503.824, Z    +0.000, E1   +39.488, E3 +82490.219}
ENDSPLINE

